Omron Sysmac Studio project 17-703_20171113_1 (Sysmac Studio 1.19.0.13, StandardProject)

# Controller new_Controller_0: NX1P2-9024DT version 1.13
Units and slaves: 節點1 : ASDA-A2-E CoE Drive (E001); 節點2 : ASDA-A2-E CoE Drive (E002)
Axis MC_Axis000, settings changed from default: AxisType=ServoType, FunctionLimit=SingleAxisPTP, UnitsConversion=EnumElement2, UnitsNumerator=1280000, UnitsDenominator=20, MaxVelocity=500, MaxJogVelocity=500, PositiveSoftwareLimit=305, HomingMode=BackupAndProximitySignalOn, StartDirection=NegativeDirection, HomingVelocity=50, HomingApproachVelocity=3, CompensationVelocity=1
Axis MC_Axis001, settings changed from default: AxisNumber=1, AxisType=ServoType, FunctionLimit=SingleAxisPTP, UnitsConversion=EnumElement2, UnitsNumerator=1280000, UnitsDenominator=20, MaxVelocity=500, MaxJogVelocity=500, PositiveSoftwareLimit=307, NegativeSoftwareLimit=-20, HomingMode=BackupAndProximitySignalOn, StartDirection=NegativeDirection, HomingVelocity=50, HomingApproachVelocity=3, CompensationVelocity=1
Task PrimaryTask (priority 4, period or condition 2000): prAxis, prConverter, prError, Postion_Control, PR_fix, 鎖付程式, 異常回0點, 系統初始, cycletime2, 原點復歸

TYPE stWorkPositionData : STRUCT
    ExPosition_X : array[0..10,0..10] of LREAL;  (* X軸鎖付位置 *)
    ExPosition_Y : array[0..10,0..10] of LREAL;  (* Y軸鎖付位置 *)
    ScrewData : array[0..10,0..10] of INT;  (* 鎖組別 *)
    Name_Data : array[0..10] of STRING[16];  (* 機種名稱 *)
    SV_AbsSpeed_X : array[0..10,0..10] of LREAL;  (* 伺服X_ABS速度32 *)
    SV_AbsSpeed_Y : array[0..10,0..10] of LREAL;  (* 伺服Y_ABS速度32 *)
    FinialPoint : array[0..10,0..10] of BOOL;
END_STRUCT END_TYPE
TYPE stAxis : STRUCT
    pbServoOn : BOOL;
    pbReset : BOOL;
    pbSerchHome : BOOL;  (* 原點搜尋開關 *)
    pbJOGForward : BOOL;  (* 手動前進 *)
    pbJOGBackward : BOOL;  (* 手動後退 *)
    pbStop : BOOL;
    pbMoveAbs : BOOL;  (* 自動移位開始 *)
    bMoveAbsDone : BOOL;  (* 到達位置 *)
    bHoming : BOOL;  (* 原點搜尋中 *)
    bServoOn : BOOL;
    bAtTHMoveSavePosition : BOOL;
    lrCurrentPosition : LREAL;  (* 現在位置 *)
    lrMoveAbsAddData : LREAL;  (* 自動移動位置 *)
    lrMoveAbsVelocity : LREAL;  (* 自動移動速度 *)
    lrMoveJogVelocity : LREAL;  (* 手動移動速度 *)
END_STRUCT END_TYPE

VAR_GLOBAL
    PB_Reset : BOOL;  (* 停止復歸開關; at BuiltInIO://cpu/#0/Input_Bit_01; published *)
    PB_Start : BOOL;  (* 啟動開關; at BuiltInIO://cpu/#0/Input_Bit_00; published *)
    PB_EStop : BOOL;  (* 急停開關; at BuiltInIO://cpu/#0/Input_Bit_02; published *)
    LS_UpDownBack : BOOL;  (* 鎖螺絲歸; at BuiltInIO://cpu/#0/Input_Bit_03; published *)
    LS_UpDownOut : BOOL;  (* 鎖螺絲出; at BuiltInIO://cpu/#0/Input_Bit_04; published *)
    LS_FixBack : BOOL;  (* 壓制歸; at BuiltInIO://cpu/#0/Input_Bit_05; published *)
    LS_FixOut : BOOL;  (* 壓制出; at BuiltInIO://cpu/#0/Input_Bit_06; published *)
    SNR_AirSource : BOOL;  (* 入氣源; at BuiltInIO://cpu/#0/Input_Bit_07; published *)
    SNR_CheckBody : BOOL;  (* 本體檢知; at BuiltInIO://cpu/#0/Input_Bit_08; published *)
    SNR_GratingUP : BOOL;  (* 安全光柵上; at BuiltInIO://cpu/#0/Input_Bit_09; published *)
    SNR_GratingDown : BOOL;  (* 安全光柵下; at BuiltInIO://cpu/#0/Input_Bit_10; published *)
    Check_GratingUP : BOOL;  (* 光柵自我檢測上; at BuiltInIO://cpu/#0/Input_Bit_11; published *)
    Check_GratingDown : BOOL;  (* 光柵自我檢測下; at BuiltInIO://cpu/#0/Input_Bit_12; published *)
    SNR_Float : BOOL;  (* 浮瑣檢知; at BuiltInIO://cpu/#0/Input_Bit_13; published *)
    SOL_FixBack : BOOL;  (* 壓制; at BuiltInIO://cpu/#0/Output_Bit_00; published *)
    SOL_UpDownBack : BOOL;  (* 鎖付上下; at BuiltInIO://cpu/#0/Output_Bit_01; published *)
    BZ : BOOL;  (* at BuiltInIO://cpu/#0/Output_Bit_02; published *)
    YL : BOOL;  (* at BuiltInIO://cpu/#0/Output_Bit_03; published *)
    GL : BOOL;  (* at BuiltInIO://cpu/#0/Output_Bit_04; published *)
    RL : BOOL;  (* at BuiltInIO://cpu/#0/Output_Bit_05; published *)
    NameTestData AT %w400 : ARRAY[0..1] OF STRING[16];
    SOL_FixOut : BOOL;  (* at BuiltInIO://cpu/#0/Output_Bit_06; published *)
    SOL_UpDownOut : BOOL;  (* at BuiltInIO://cpu/#0/Output_Bit_07; published *)
    Servo_OUT_Ready : BOOL;  (* 日東準備; at IOBus://unit#2/Input Bit 16 bits/Input Bit 00; published *)
    Servo_OUT_OK : BOOL;  (* 日東鎖付OK; at IOBus://unit#2/Input Bit 16 bits/Input Bit 01; published *)
    Servo_OUT_NOK : BOOL;  (* 日東鎖付NG; at IOBus://unit#2/Input Bit 16 bits/Input Bit 02; published *)
    Servo_OUT_Error : BOOL;  (* 日東異常; at IOBus://unit#2/Input Bit 16 bits/Input Bit 03; published *)
    Servo_OUT_Fioat : BOOL;  (* 日東鎖螺絲浮鎖測試OK; at IOBus://unit#2/Input Bit 16 bits/Input Bit 04; published *)
    Servo_OUT_Start : BOOL;  (* 日東同期鎖付啟動; at IOBus://unit#2/Input Bit 16 bits/Input Bit 05; published *)
    Servo_OUT_Angle : BOOL;  (* 日東角度判定OK; at IOBus://unit#2/Input Bit 16 bits/Input Bit 06; published *)
    Servo_OUT_Wave_AX1 : BOOL;  (* 日東波形處理OK; at IOBus://unit#2/Input Bit 16 bits/Input Bit 07; published *)
    Servo_IN_Start : BOOL;  (* 日東啟動; at IOBus://unit#3/Output Bit 8 bits/Output Bit 00; published *)
    Servo_IN_TorqueBit0 : BOOL;  (* 日東工作選擇0; at IOBus://unit#3/Output Bit 8 bits/Output Bit 01; published *)
    Servo_IN_TorqueBit1 : BOOL;  (* 日東工作選擇1; at IOBus://unit#3/Output Bit 8 bits/Output Bit 02; published *)
    Servo_IN_TorqueBit2 : BOOL;  (* 日東工作選擇2; at IOBus://unit#3/Output Bit 8 bits/Output Bit 03; published *)
    Servo_IN_TorqueBit3 : BOOL;  (* 日東工作選擇3; at IOBus://unit#3/Output Bit 8 bits/Output Bit 04; published *)
    Servo_IN_output : BOOL;  (* 日東外部信號; at IOBus://unit#3/Output Bit 8 bits/Output Bit 05; published *)
    Servo_IN_ALLStart : BOOL;  (* 日東同期鎖付啟動; at IOBus://unit#3/Output Bit 8 bits/Output Bit 06; published *)
END_VAR
VAR_GLOBAL CONSTANT
    MC_Axis000 : _sAXIS_REF;  (* at MC://_MC_AX[0] *)
    MC_Axis001 : _sAXIS_REF;  (* at MC://_MC_AX[1] *)
END_VAR
VAR_GLOBAL
    Ax_X : stAxis;
    Ax_Y : stAxis;
END_VAR
VAR_GLOBAL RETAIN
    WorkPositionData : stWorkPositionData;  (* published *)
END_VAR
VAR_GLOBAL
    SystemReadyStatus : BOOL;  (* published *)
    MachineRun : BOOL;  (* published *)
    ErrorStatus_MachineStop : BOOL;  (* 機器停機異常; published *)
    ErrorStatus_MachineNonStop : BOOL;  (* 機器不停機異常; published *)
    Manual2AutoFlag : BOOL;  (* published *)
    AutoStatus AT %W000.00 : BOOL;  (* 自動狀態; published *)
    PB_UpDownBack AT %W000.01 : BOOL;  (* 手動鎖付上; published *)
    PB_UpDownOut AT %W000.02 : BOOL;  (* 手動鎖付下; published *)
    PB_FixBack AT %W000.03 : BOOL;  (* 手動壓制回; published *)
    PB_FixOut AT %W000.04 : BOOL;  (* 手動壓制出; published *)
    PB_ScrewStart AT %W000.05 : BOOL;  (* published *)
    PB_ServoY_Back AT %W000.06 : BOOL;  (* 手動伺服Y回; published *)
    PB_ServoY_Out AT %W000.07 : BOOL;  (* 手動伺服Y出; published *)
    PB_ServoX_Back AT %W000.08 : BOOL;  (* 手動伺服X回; published *)
    PB_ServoX_Out AT %W000.09 : BOOL;  (* 手動伺服X出; published *)
    PB_ServoOn_X AT %W000.10 : BOOL;  (* 手動伺服X_ServoON; published *)
    PB_ServoOn_Y AT %W000.11 : BOOL;  (* 手動伺服Y_ServoON; published *)
    PB_SetPostion AT %W000.12 : BOOL;  (* 位置設定開關; published *)
    PB_FinalPoint AT %W000.13 : BOOL;  (* 最終點設定開關; published *)
    PB_PostionGo AT %W000.14 : BOOL;  (* 點位啟動; published *)
    PB_Set_Homed AT %W000.15 : BOOL;  (* 伺服回原點開關; published *)
    PB_HMI_RESRT AT %W001.00 : BOOL;  (* published *)
    State_Homed_MC AT %W001.01 : BOOL;  (* 伺服原點; published *)
    State_Homing_MC AT %W001.02 : BOOL;  (* 伺服回原點中; published *)
    State_HomeSerching_X AT %W001.03 : BOOL;  (* X伺服回原點中; published *)
    State_Homed_X AT %W001.04 : BOOL;  (* X伺服原點; published *)
    State_HomeSerching_Y AT %W001.05 : BOOL;  (* Y伺服回原點中; published *)
    State_Homed_Y AT %W001.06 : BOOL;  (* Y伺服原點; published *)
    ScrewStartStatus AT %W001.07 : BOOL;  (* published *)
    LS_FixOut1 AT %W001.15 : BOOL;  (* published *)
    HMI_ScrewOK1 AT %W002.00 : BOOL;  (* published *)
    HMI_ScrewOK2 AT %W002.01 : BOOL;  (* published *)
    LS_FixBack1 AT %W001.14 : BOOL;  (* published *)
    LS_UpDownBack1 AT %W001.12 : BOOL;  (* published *)
    PB_HMI_SetScrew AT %w001.11 : BOOL;  (* published *)
    LS_UpDownOut1 AT %W001.13 : BOOL;  (* published *)
    PB_HMI_BzStpo AT %w001.10 : BOOL;  (* published *)
    ScrewFinish AT %W001.08 : BOOL;  (* published *)
    HMI_Servo_IN_Start AT %W001.09 : BOOL;  (* published *)
END_VAR
VAR_GLOBAL RETAIN
    SV_ServoXJogSpeed : LREAL;  (* 設定伺服X_JOG速度64; published *)
    SV_ServoYJogSpeed : LREAL;  (* 設定伺服Y_JOG速度64; published *)
    SV_ServoXJogSpeed_R AT %D000 : REAL;  (* 設定伺服X_JOG速度32; published *)
    SV_ServoYJogSpeed_R AT %D002 : REAL;  (* 設定伺服Y_JOG速度32; published *)
    SV_AbsSpeedX_R AT %D004 : REAL;  (* 設定伺服X_ABS速度32; published *)
    SV_AbsSpeedY_R AT %D006 : REAL;  (* 設定伺服Y_ABS速度32; published *)
    HMI_SV_AbsSpeedX_R AT %D008 : REAL;  (* 顯示伺服X_ABS速度32; published *)
    HMI_SV_AbsSpeedY_R AT %D010 : REAL;  (* 顯示伺服Y_ABS速度32; published *)
    HMI_SV_CurrentPositionX AT %D012 : REAL;  (* 人機現在位置X顯示; published *)
    HMI_SV_CurrentPositionY AT %D014 : REAL;  (* 人機現在位置Y顯示; published *)
    Type_Data AT %D042 : INT;  (* 設定組別; published *)
    PointData AT %D043 : INT;  (* 設定點位; published *)
    Screw_Data1 AT %D044 : INT;  (* 設定鎖付值; published *)
    Screw_Data2 AT %D045 : INT;
    Screw_Data3 AT %D046 : INT;
    Screw_Data4 AT %D047 : INT;
    OK_Count AT %D050 : DINT;  (* published *)
    AllOK_Count AT %D052 : DINT;  (* published *)
    HMISV_CycleTime1 AT %D054 : DINT;  (* published *)
    HMISV_CycleTime2 AT %D056 : DINT;  (* published *)
END_VAR
VAR_GLOBAL
    HMI_Name : ARRAY[0..10] OF STRING[32];  (* 顯示已設定組別名稱; published *)
    HMI_ScrewOK3 AT %W002.02 : BOOL;  (* published *)
    HMI_ScrewOK4 AT %W002.03 : BOOL;  (* published *)
END_VAR
VAR_GLOBAL RETAIN
    HMI_Name1 AT %D200 : STRING[16];  (* published *)
    HMI_Name2 AT %D208 : STRING[16];  (* published *)
    HMI_Name3 AT %D216 : STRING[16];  (* published *)
    HMI_Name4 AT %D224 : STRING[16];  (* published *)
    HMI_Name5 AT %D232 : STRING[16];  (* published *)
    HMI_Name6 AT %D240 : STRING[16];  (* published *)
    HMI_Name7 AT %D248 : STRING[16];  (* published *)
    HMI_Name8 AT %D256 : STRING[16];  (* published *)
    HMI_Name9 AT %D264 : STRING[16];  (* published *)
    HMI_Name10 AT %D272 : STRING[16];  (* published *)
END_VAR
VAR_GLOBAL
    HMI_SV_Name AT %W360 : STRING[16];  (* published *)
    HMI_ScrewNG1 AT %W002.04 : BOOL;  (* published *)
    HMI_ScrewNG2 AT %W002.05 : BOOL;  (* published *)
    HMI_ScrewNG3 AT %W002.06 : BOOL;  (* published *)
    HMI_ScrewNG4 AT %W002.07 : BOOL;  (* published *)
    HMI_Float1 AT %W002.08 : BOOL;  (* published *)
    HMI_SV_Screw_Data4 AT %W153 : INT;
    HMI_SV_Screw_Data3 AT %W152 : INT;
    HMI_SV_Screw_Data2 AT %W151 : INT;
    HMI_SV_Screw_Data1 AT %W150 : INT;
    HMI_SV_Screw_Data AT %W104 : INT;  (* 顯示現在鎖付值; published *)
    HMI_PositionY AT %W102 : REAL;  (* 顯示已設定位置Y顯示; published *)
    HMI_PositionX AT %W100 : REAL;  (* 顯示已設定位置X顯示; published *)
    HMI_Float2 AT %W002.09 : BOOL;  (* published *)
    HMI_Float4 AT %W002.11 : BOOL;  (* published *)
    HMI_SVFinalPoint AT %W002.12 : BOOL;  (* HMI最終點顯示; published *)
    PB_ResetOk_Count AT %W002.13 : BOOL;  (* published *)
    PB_Name_Set AT %w002.14 : BOOL;  (* published *)
    HMI_Float3 AT %W002.10 : BOOL;  (* published *)
END_VAR
VAR_GLOBAL RETAIN
    Screw_OK : ARRAY[0..10] OF BOOL;  (* published *)
    Screw_NG : ARRAY[0..10] OF BOOL;  (* published *)
    Screw_Float : ARRAY[0..10] OF BOOL;  (* published *)
END_VAR
VAR_GLOBAL
    Error_LS_UpDownBack AT %W200.00 : BOOL;  (* published *)
    Error_LS_UpDownOut AT %W200.01 : BOOL;  (* published *)
    Error_LS_FixBack AT %W200.02 : BOOL;  (* published *)
    Error_LS_FixOut AT %W200.03 : BOOL;  (* published *)
    Error_Check_GratingUP AT %W200.04 : BOOL;  (* 光柵自我檢測上異常; published *)
    Error_Check_GratingDown AT %W200.05 : BOOL;  (* 光柵自我檢測下異常; published *)
    Error_GratingUP AT %W200.06 : BOOL;  (* 光柵上異常; published *)
    Error_GratingDown AT %W200.07 : BOOL;  (* 光柵下異常; published *)
    Error_EStopPB AT %W200.08 : BOOL;  (* published *)
    Error_ChangeBodyNG AT %W200.14 : BOOL;  (* published *)
    Error_ScrewNG AT %W200.13 : BOOL;  (* published *)
    Error_SNR_CheckBody AT %W200.12 : BOOL;  (* published *)
    Error_SNR_AirSource AT %W200.11 : BOOL;  (* published *)
    Error_Servo_Y AT %W200.10 : BOOL;  (* 伺服異常Y; published *)
    Error_Servo_X AT %W200.09 : BOOL;  (* 伺服異常X; published *)
    Error_LS_Status : BOOL;  (* 磁簧開關異常; published *)
    Error_Grating_Status : BOOL;  (* published *)
    Error_Status : BOOL;  (* published *)
    Error_Servo : BOOL;  (* published *)
    XN_OT : BOOL;  (* published *)
    XP_OT : BOOL;  (* published *)
    YN_OT : BOOL;  (* published *)
    YP_OT : BOOL;  (* published *)
    MachineRunStatus : BOOL;
    HMI_LT_ServoRuning AT %W003.01 : BOOL;  (* published *)
    HMI_LT_ServoFinish AT %w003.00 : BOOL;  (* published *)
    LT_ServoFinish1 AT %w003.02 : BOOL;  (* published *)
    LT_ServoFinish2 AT %w003.04 : BOOL;  (* published *)
    LT_ServoRuning1 AT %w003.05 : BOOL;  (* published *)
    LT_ServoRuning2 AT %w003.06 : BOOL;  (* published *)
    Error_XP_OT AT %W200.15 : BOOL;  (* published *)
    Error_XN_OT AT %W201.00 : BOOL;  (* published *)
    Error_YP_OT AT %W201.01 : BOOL;  (* published *)
    Error_YN_OT AT %W201.02 : BOOL;  (* published *)
END_VAR
VAR_GLOBAL RETAIN
    Screw_Data5 AT %D060 : INT;  (* published *)
    Screw_Data6 AT %D061 : INT;  (* published *)
    Screw_Data7 AT %D062 : INT;  (* published *)
    Screw_Data8 AT %D063 : INT;  (* published *)
    Screw_Data9 AT %D064 : INT;  (* published *)
    Screw_Data10 AT %D065 : INT;  (* published *)
END_VAR
VAR_GLOBAL
    HMI_SV_Screw_Data5 AT %W154 : INT;  (* published *)
    HMI_SV_Screw_Data6 AT %W155 : INT;  (* published *)
    HMI_SV_Screw_Data7 AT %W156 : INT;  (* published *)
    HMI_SV_Screw_Data8 AT %W157 : INT;  (* published *)
    HMI_SV_Screw_Data9 AT %W158 : INT;  (* published *)
    HMI_SV_Screw_Data10 AT %W159 : INT;  (* published *)
    LS_ExternalStart : BOOL;  (* 外部可啟動信號; at IOBus://unit#2/Input Bit 16 bits/Input Bit 08; published *)
    HMI_SV_ReclaimerOK AT %w003.07 : BOOL;  (* 外部取料完成; published *)
END_VAR
VAR_GLOBAL RETAIN
    ReclaimerOK : BOOL;  (* published *)
END_VAR
VAR_GLOBAL
    Error_ReclaimerOK AT %W201.03 : BOOL;  (* 取料未完成異常; published *)
END_VAR
VAR_GLOBAL RETAIN
    PB_ExternalStart AT %H00.0 : BOOL;  (* published *)
END_VAR

PROGRAM prAxis
VAR
    MC_Power_Ax1 : MC_Power;
    MC_Power_Ax2 : MC_Power;
    MC_Home_Ax1 : MC_Home;
    MC_Home_Ax2 : MC_Home;
    MC_MoveJog_Ax1 : MC_MoveJog;
    MC_MoveJog_Ax2 : MC_MoveJog;
    MC_Reset_Ax1 : MC_Reset;
    MC_Reset_Ax2 : MC_Reset;
    MC_MoveAbsolute_Ax1 : MC_MoveAbsolute;
    MC_MoveAbsolute_Ax2 : MC_MoveAbsolute;
    MC_Stop_Ax1 : MC_Stop;
    MC_Stop_Ax2 : MC_Stop;
    XN_HOME : BOOL;
    Y_HOME : BOOL;
END_VAR
VAR_EXTERNAL CONSTANT
    MC_Axis001 : _sAXIS_REF;
END_VAR
VAR_EXTERNAL
    Ax_X : stAxis;
END_VAR
VAR_EXTERNAL CONSTANT
    MC_Axis000 : _sAXIS_REF;
END_VAR
VAR_EXTERNAL
    Ax_Y : stAxis;
    WorkPositionData : stWorkPositionData;
    PB_EStop : BOOL;
    Error_EStopPB : BOOL;
    PB_ServoOn_X : BOOL;
    PB_ServoOn_Y : BOOL;
    PB_Reset : BOOL;
    XP_OT : BOOL;
    XN_OT : BOOL;
    YN_OT : BOOL;
    YP_OT : BOOL;
    ErrorStatus_MachineStop : BOOL;
    LS_UpDownBack : BOOL;
    SOL_UpDownOut : BOOL;
    LS_UpDownBack1 : BOOL;
    SNR_AirSource : BOOL;
    SNR_GratingDown : BOOL;
    SNR_GratingUP : BOOL;
    Error_GratingUP : BOOL;
    Error_GratingDown : BOOL;
    Error_Grating_Status : BOOL;
    Error_XP_OT : BOOL;
    Error_YP_OT : BOOL;
    Error_YN_OT : BOOL;
END_VAR
(*X軸*)
//Servo on
Ax_X.pbServoOn:=PB_ServoOn_X;
MC_Power_Ax1(Axis:=MC_Axis000, Enable:=Ax_X.pbServoOn AND NOT(Error_EStopPB));
//Reset
MC_Reset_Ax1(Axis:=MC_Axis000, Execute:=Ax_X.pbReset);
//Home
MC_Home_Ax1(Axis:=MC_Axis000, Execute:=Ax_X.pbSerchHome AND Ax_X.bServoOn);
//STOP
MC_Stop_Ax1(Axis:=MC_Axis000, Execute:=Ax_X.pbStop);
//JOG
MC_MoveJog_Ax1(Axis:=MC_Axis000, PositiveEnable:=Ax_X.pbJOGForward , NegativeEnable:=Ax_X.pbJOGBackward , Velocity:=Ax_X.lrMoveJogVelocity,acceleration:=5000,deceleration:=5000);
//絕對定位
MC_MoveAbsolute_Ax1(Axis:=MC_Axis000, Execute:=Ax_X.pbMoveAbs AND Ax_X.bServoOn AND MC_Axis000.Details.Homed,
					Position:=Ax_X.lrMoveAbsAddData,	Velocity:=Ax_X.lrMoveAbsVelocity,acceleration:=5000,deceleration:=5000,
					Done=>Ax_X.bMoveAbsDone);

//定義
//Servo On
Ax_X.bServoOn:=MC_Axis000.DrvStatus.ServoOn;
//找HOME
Ax_X.bHoming:=MC_Axis000.Status.Homing;
//現在位置
Ax_X.lrCurrentPosition:=MC_Axis000.Act.Pos;
(*Y軸*)
//Servo on
Ax_Y.pbServoOn:=PB_ServoOn_Y;
MC_Power_Ax2(Axis:=MC_Axis001, Enable:=Ax_Y.pbServoOn AND NOT(Error_EStopPB));
//Reset
MC_Reset_Ax2(Axis:=MC_Axis001, Execute:=Ax_Y.pbReset);
//Home
MC_Home_Ax2(Axis:=MC_Axis001, Execute:=Ax_Y.pbSerchHome AND Ax_Y.bServoOn);
//STOP
MC_Stop_Ax2(Axis:=MC_Axis001, Execute:=Ax_Y.pbStop );
//JOG
MC_MoveJog_Ax2(Axis:=MC_Axis001, PositiveEnable:=Ax_Y.pbJOGForward  , NegativeEnable:=Ax_Y.pbJOGBackward  , Velocity:=Ax_Y.lrMoveJogVelocity,acceleration:=5000,deceleration:=5000);
//絕對定位
MC_MoveAbsolute_Ax2(Axis:=MC_Axis001, Execute:=Ax_Y.pbMoveAbs AND Ax_Y.bServoOn AND MC_Axis001.Details.Homed,
					Position:=Ax_Y.lrMoveAbsAddData,	Velocity:=Ax_Y.lrMoveAbsVelocity,acceleration:=5000,deceleration:=5000,
					Done=>Ax_Y.bMoveAbsDone);

//定義
//Servo On
Ax_Y.bServoOn:=MC_Axis001.DrvStatus.ServoOn;
//找HOME
Ax_Y.bHoming:=MC_Axis001.Status.Homing;
//現在位置
Ax_Y.lrCurrentPosition:=MC_Axis001.Act.Pos;

//RESET
Ax_X.pbReset:=PB_Reset;
Ax_Y.pbReset:=PB_Reset;
//Stop
Ax_X.pbStop:= NOT(PB_EStop) OR Error_Grating_Status;
Ax_Y.pbStop:= NOT(PB_EStop) OR Error_Grating_Status;
XN_OT:=MC_Axis000.DrvStatus.N_OT;
XP_OT:=MC_Axis000.DrvStatus.P_OT;
YN_OT:=MC_Axis001.DrvStatus.N_OT;
YP_OT:=MC_Axis001.DrvStatus.P_OT;
XN_HOME:=MC_Axis000.DrvStatus.HomeSw;
Y_HOME:=MC_Axis001.DrvStatus.HomeSw;
END_PROGRAM

PROGRAM prConverter
VAR
    Status_FinalPoint : BOOL;
    R_TRIG_1 : R_TRIG;
END_VAR
VAR_EXTERNAL
    SV_ServoXJogSpeed : LREAL;
    SV_AbsSpeedX_R : REAL;
    SV_ServoXJogSpeed_R : REAL;
    SV_ServoYJogSpeed : LREAL;
    SV_ServoYJogSpeed_R : REAL;
    Ax_X : stAxis;
    Type_Data : INT;
    PointData : INT;
    WorkPositionData : stWorkPositionData;
    SV_AbsSpeedY_R : REAL;
    State_Homed_X : BOOL;
END_VAR
VAR_EXTERNAL CONSTANT
    MC_Axis000 : _sAXIS_REF;
END_VAR
VAR_EXTERNAL
    State_Homed_Y : BOOL;
END_VAR
VAR_EXTERNAL CONSTANT
    MC_Axis001 : _sAXIS_REF;
END_VAR
VAR_EXTERNAL
    State_HomeSerching_X : BOOL;
    State_HomeSerching_Y : BOOL;
    Ax_Y : stAxis;
    State_Homed_MC : BOOL;
    State_Homing_MC : BOOL;
    PB_SetPostion : BOOL;
    PB_FinalPoint : BOOL;
    HMI_SV_CurrentPositionX : REAL;
    HMI_SV_CurrentPositionY : REAL;
    HMI_PositionX : REAL;
    HMI_PositionY : REAL;
    HMI_SVFinalPoint : BOOL;
    AutoStatus : BOOL;
    HMI_SV_Screw_Data : INT;
    HMI_SV_AbsSpeedX_R : REAL;
    HMI_SV_AbsSpeedY_R : REAL;
    HMI_ScrewNG1 : BOOL;
    Screw_NG : ARRAY[0..10] OF BOOL;
    HMI_ScrewNG2 : BOOL;
    HMI_ScrewNG3 : BOOL;
    HMI_ScrewNG4 : BOOL;
    HMI_ScrewOK1 : BOOL;
    Screw_OK : ARRAY[0..10] OF BOOL;
    HMI_ScrewOK2 : BOOL;
    HMI_ScrewOK3 : BOOL;
    HMI_ScrewOK4 : BOOL;
    HMI_Name1 : STRING[16];
    HMI_Name2 : STRING[16];
    HMI_Name3 : STRING[16];
    HMI_Name4 : STRING[16];
    HMI_Name5 : STRING[16];
    HMI_Name6 : STRING[16];
    HMI_Name7 : STRING[16];
    HMI_Name8 : STRING[16];
    HMI_Name9 : STRING[16];
    HMI_Name10 : STRING[16];
    HMI_Name : ARRAY[0..10] OF STRING[32];
    PB_Name_Set : BOOL;
    Screw_Data1 : INT;
    Screw_Data2 : INT;
    Screw_Data3 : INT;
    Screw_Data4 : INT;
    HMI_SV_Screw_Data1 : INT;
    HMI_SV_Screw_Data4 : INT;
    HMI_SV_Screw_Data3 : INT;
    HMI_SV_Screw_Data2 : INT;
    PB_HMI_SetScrew : BOOL;
    HMI_SV_Name : STRING[16];
    HMISV_CycleTime1 : DINT;
    NameTestData : ARRAY[0..1] OF STRING[16];
    Screw_Data10 : INT;
    Screw_Data9 : INT;
    Screw_Data5 : INT;
    Screw_Data6 : INT;
    Screw_Data7 : INT;
    Screw_Data8 : INT;
    HMI_SV_Screw_Data10 : INT;
    HMI_SV_Screw_Data9 : INT;
    HMI_SV_Screw_Data8 : INT;
    HMI_SV_Screw_Data7 : INT;
    HMI_SV_Screw_Data6 : INT;
    HMI_SV_Screw_Data5 : INT;
    HMI_SV_ReclaimerOK : BOOL;
    ReclaimerOK : BOOL;
    LS_ExternalStart : BOOL;
    Screw_Float : ARRAY[0..10] OF BOOL;
    HMI_Float2 : BOOL;
    HMI_Float3 : BOOL;
    HMI_Float4 : BOOL;
    HMI_Float1 : BOOL;
END_VAR
SV_ServoXJogSpeed:=REAL_TO_LREAL(SV_ServoXJogSpeed_R);//X軸手動速度單位轉換
SV_ServoYJogSpeed:=REAL_TO_LREAL(SV_ServoYJogSpeed_R);//Y軸手動速度單位轉換
State_Homed_X:=MC_Axis000.Details.Homed;//X軸復歸完成
State_Homed_Y:=MC_Axis001.Details.Homed;//Y軸復歸完成
State_HomeSerching_X:=Ax_X.bHoming;//X軸復歸中
State_HomeSerching_Y:=Ax_Y.bHoming;//Y軸復歸中
State_Homed_MC:=State_Homed_X AND State_Homed_Y AND NOT(State_Homing_MC);//原點復歸完成
State_Homing_MC:=State_HomeSerching_X OR State_HomeSerching_Y;//原點復歸中
//位置_鎖付組別寫入
IF PB_SetPostion THEN
	WorkPositionData.ExPosition_X[Type_Data,PointData]:=Ax_X.lrCurrentPosition;
    WorkPositionData.ExPosition_Y[Type_Data,PointData]:=Ax_Y.lrCurrentPosition;
	WorkPositionData.SV_AbsSpeed_X[Type_Data,PointData]:=REAL_TO_LREAL(SV_AbsSpeedX_R);
    WorkPositionData.SV_AbsSpeed_Y[Type_Data,PointData]:=REAL_TO_LREAL(SV_AbsSpeedY_R);
END_IF;

//最終點寫入
R_TRIG_1(Clk:=PB_FinalPoint);
IF R_TRIG_1.Q AND NOT(Status_FinalPoint)  THEN
	WorkPositionData.FinialPoint[Type_Data,PointData]:=TRUE;
END_IF;
//最終點取消
IF R_TRIG_1.Q AND Status_FinalPoint  THEN
	WorkPositionData.FinialPoint[Type_Data,PointData]:=FALSE;
END_IF;
Status_FinalPoint:=WorkPositionData.FinialPoint[Type_Data,PointData];

//現在位置HMI
HMI_SV_CurrentPositionX:=LREAL_TO_REAL(Ax_X.lrCurrentPosition);
HMI_SV_CurrentPositionY:=LREAL_TO_REAL(Ax_Y.lrCurrentPosition);
//設定位置
HMI_PositionX:=LREAL_TO_REAL(WorkPositionData.ExPosition_X[Type_Data,PointData]);
HMI_PositionY:=LREAL_TO_REAL(WorkPositionData.ExPosition_Y[Type_Data,PointData]);
//最終點顯示
HMI_SVFinalPoint:=WorkPositionData.FinialPoint[Type_Data,PointData];
//人機顯示
HMI_SV_AbsSpeedX_R:=LREAL_TO_REAL(WorkPositionData.SV_AbsSpeed_X[Type_Data,PointData]);
HMI_SV_AbsSpeedY_R:=LREAL_TO_REAL(WorkPositionData.SV_AbsSpeed_Y[Type_Data,PointData]);
//HMI_Name[Type_Data]:=WorkPositionData.Name_Data[Type_Data];
HMI_SV_Name:=WorkPositionData.Name_Data[Type_Data];
NameTestData[0]:=HMI_SV_Name;
HMI_ScrewNG1:=Screw_NG[1];
HMI_ScrewNG2:=Screw_NG[2];
HMI_ScrewNG3:=Screw_NG[3];
HMI_ScrewNG4:=Screw_NG[4];
HMI_ScrewOK1:=Screw_OK[1];
HMI_ScrewOK2:=Screw_OK[2];
HMI_ScrewOK3:=Screw_OK[3];
HMI_ScrewOK4:=Screw_OK[4];
HMI_Float1:=Screw_Float[1];
HMI_Float2:=Screw_Float[2];
HMI_Float3:=Screw_Float[3];
HMI_Float4:=Screw_Float[4];
IF PB_Name_Set THEN
WorkPositionData.Name_Data[1]:=HMI_Name1;
WorkPositionData.Name_Data[2]:=HMI_Name2;
WorkPositionData.Name_Data[3]:=HMI_Name3;
WorkPositionData.Name_Data[4]:=HMI_Name4;
WorkPositionData.Name_Data[5]:=HMI_Name5;
WorkPositionData.Name_Data[6]:=HMI_Name6;
WorkPositionData.Name_Data[7]:=HMI_Name7;
WorkPositionData.Name_Data[8]:=HMI_Name8;
WorkPositionData.Name_Data[9]:=HMI_Name9;
WorkPositionData.Name_Data[10]:=HMI_Name10;
END_IF;
//日東組別寫入
IF PB_HMI_SetScrew THEN
WorkPositionData.ScrewData[Type_Data,1]:=Screw_Data1;
WorkPositionData.ScrewData[Type_Data,2]:=Screw_Data2;
WorkPositionData.ScrewData[Type_Data,3]:=Screw_Data3;
WorkPositionData.ScrewData[Type_Data,4]:=Screw_Data4;
WorkPositionData.ScrewData[Type_Data,5]:=Screw_Data5;
WorkPositionData.ScrewData[Type_Data,6]:=Screw_Data6;
WorkPositionData.ScrewData[Type_Data,7]:=Screw_Data7;
WorkPositionData.ScrewData[Type_Data,8]:=Screw_Data8;
WorkPositionData.ScrewData[Type_Data,9]:=Screw_Data9;
WorkPositionData.ScrewData[Type_Data,10]:=Screw_Data10;
END_IF;

//日東組別顯示
HMI_SV_Screw_Data:=WorkPositionData.ScrewData[Type_Data,PointData];
HMI_SV_Screw_Data1:=WorkPositionData.ScrewData[Type_Data,1];
HMI_SV_Screw_Data2:=WorkPositionData.ScrewData[Type_Data,2];
HMI_SV_Screw_Data3:=WorkPositionData.ScrewData[Type_Data,3];
HMI_SV_Screw_Data4:=WorkPositionData.ScrewData[Type_Data,4];
HMI_SV_Screw_Data5:=WorkPositionData.ScrewData[Type_Data,5];
HMI_SV_Screw_Data6:=WorkPositionData.ScrewData[Type_Data,6];
HMI_SV_Screw_Data7:=WorkPositionData.ScrewData[Type_Data,7];
HMI_SV_Screw_Data8:=WorkPositionData.ScrewData[Type_Data,8];
HMI_SV_Screw_Data9:=WorkPositionData.ScrewData[Type_Data,9];
HMI_SV_Screw_Data10:=WorkPositionData.ScrewData[Type_Data,10];
//外部取料信號顯示
HMI_SV_ReclaimerOK:=ReclaimerOK;	
END_PROGRAM

PROGRAM prError
VAR
    TON1 : ARRAY[0..10] OF TON;
    ExternalStart_status : BOOL;
    R_TRIG_1 : R_TRIG;
    R_TRIG_2 : R_TRIG;
    F_TRIG_1 : R_TRIG;
    F_TRIG_2 : F_TRIG;
END_VAR
VAR_EXTERNAL
    AutoStatus : BOOL;
    PB_Reset : BOOL;
    LS_UpDownBack : BOOL;
    SOL_UpDownBack : BOOL;
    LS_UpDownOut : BOOL;
    Error_LS_UpDownBack : BOOL;
    SOL_UpDownOut : BOOL;
    Error_LS_UpDownOut : BOOL;
    SOL_FixBack : BOOL;
    LS_FixBack : BOOL;
    Error_LS_FixBack : BOOL;
    LS_FixOut : BOOL;
    SOL_FixOut : BOOL;
    Error_LS_FixOut : BOOL;
    Error_EStopPB : BOOL;
    PB_EStop : BOOL;
END_VAR
VAR_EXTERNAL CONSTANT
    MC_Axis000 : _sAXIS_REF;
END_VAR
VAR_EXTERNAL
    Error_Servo_X : BOOL;
END_VAR
VAR_EXTERNAL CONSTANT
    MC_Axis001 : _sAXIS_REF;
END_VAR
VAR_EXTERNAL
    Error_Servo_Y : BOOL;
    Check_GratingUP : BOOL;
    Error_Check_GratingUP : BOOL;
    Check_GratingDown : BOOL;
    Error_Check_GratingDown : BOOL;
    SystemReadyStatus : BOOL;
    MachineRun : BOOL;
    SNR_GratingUP : BOOL;
    Error_GratingUP : BOOL;
    SNR_GratingDown : BOOL;
    Error_GratingDown : BOOL;
    SNR_AirSource : BOOL;
    Error_SNR_AirSource : BOOL;
    ErrorStatus_MachineStop : BOOL;
    Error_LS_Status : BOOL;
    Error_Servo : BOOL;
    Servo_OUT_Error : BOOL;
    Error_Grating_Status : BOOL;
    SNR_CheckBody : BOOL;
    Error_SNR_CheckBody : BOOL;
    PB_HMI_RESRT : BOOL;
    MachineRunStatus : BOOL;
    Screw_NG : ARRAY[0..10] OF BOOL;
    Error_ScrewNG : BOOL;
    LS_UpDownBack1 : BOOL;
    LS_UpDownOut1 : BOOL;
    LS_FixBack1 : BOOL;
    LS_FixOut1 : BOOL;
    Servo_IN_ALLStart : BOOL;
    Servo_IN_Start : BOOL;
    HMI_Servo_IN_Start : BOOL;
    ScrewFinish : BOOL;
    Error_ChangeBodyNG : BOOL;
    PB_Start : BOOL;
    Ax_X : stAxis;
    Ax_Y : stAxis;
    HMI_LT_ServoFinish : BOOL;
    LT_ServoFinish1 : BOOL;
    LT_ServoFinish2 : BOOL;
    HMI_LT_ServoRuning : BOOL;
    LT_ServoRuning1 : BOOL;
    LT_ServoRuning2 : BOOL;
    Type_Data : INT;
    WorkPositionData : stWorkPositionData;
    XP_OT : BOOL;
    Error_XP_OT : BOOL;
    PB_ServoOn_X : BOOL;
    XN_OT : BOOL;
    YP_OT : BOOL;
    Error_YP_OT : BOOL;
    PB_ServoOn_Y : BOOL;
    YN_OT : BOOL;
    Error_YN_OT : BOOL;
    Error_XN_OT : BOOL;
    State_Homed_MC : BOOL;
    LS_ExternalStart : BOOL;
    ReclaimerOK : BOOL;
    Error_ReclaimerOK : BOOL;
    PB_ExternalStart : BOOL;
    Screw_Float : ARRAY[0..10] OF BOOL;
END_VAR
IF AutoStatus AND NOT(PB_Reset) AND Type_Data<10  THEN
    TON1[0](In:=((SOL_UpDownBack AND NOT(LS_UpDownBack)) OR (NOT(LS_UpDownBack)  AND NOT(LS_UpDownOut) ) ), PT:=T#2s);
 (*上下歸異常磁簧開關*)
   IF TON1[0].Q THEN
	   Error_LS_UpDownBack:=TRUE;
   END_IF;
   IF LS_UpDownBack THEN
	   SOL_UpDownBack:=FALSE;
   END_IF;
  TON1[1](In:=((SOL_UpDownOut AND NOT(LS_UpDownOut)) OR (NOT(LS_UpDownBack) AND NOT(LS_UpDownOut) )  ), PT:=T#2s);
  (*上下出異常磁簧開關*)
   IF TON1[1].Q THEN
	   Error_LS_UpDownOut:=TRUE;
   END_IF;
   IF LS_UpDownOut THEN
	   SOL_UpDownOut:=FALSE;
   END_IF;
   TON1[2](In:=((SOL_FixBack AND NOT(LS_FixBack)) OR (NOT(LS_FixBack) AND NOT(LS_FixOut) )  ), PT:=T#2s);
 (*壓制歸異常磁簧開關*)
   IF TON1[2].Q THEN
	   Error_LS_FixBack:=TRUE;
   END_IF;
   IF LS_FixBack THEN
	   SOL_FixBack:=FALSE;
   END_IF;
TON1[3](In:=((SOL_FixOut AND NOT(LS_FixOut)) OR (NOT(LS_FixBack) AND NOT(LS_FixOut) ) ), PT:=T#2s);
(*壓制出異常磁簧開關*)
   IF TON1[3].Q THEN
	   Error_LS_FixOut:=TRUE;
   END_IF;
   IF LS_FixOut THEN
	   SOL_FixOut:=FALSE;
   END_IF;
END_IF;

//ESTOP
TON1[4](In:=P_On , PT:=T#100ms);
IF TON1[4].Q AND NOT(PB_EStop)   THEN
	Error_EStopPB:=TRUE;
END_IF;

//氣壓源異常
IF NOT(SNR_AirSource) AND TON1[4].Q THEN
	Error_SNR_AirSource:=TRUE;
END_IF;

//SERVO
IF MC_Axis000.DrvStatus.DrvAlarm AND TON1[4].Q THEN
	Error_Servo_X:=TRUE;
END_IF;
IF MC_Axis001.DrvStatus.DrvAlarm AND TON1[4].Q THEN
	Error_Servo_Y:=TRUE;
END_IF;

//本體異常
R_TRIG_1(Clk:=MachineRun);
IF R_TRIG_1.Q AND NOT(SNR_CheckBody) AND NOT(Type_Data=10) THEN
	Error_SNR_CheckBody:=TRUE;
END_IF;

//光閘自我檢測異常(上)
//IF NOT(Check_GratingUP) AND TON1[4].Q  THEN
//	Error_Check_GratingUP:=TRUE;
//END_IF;

//光閘自我檢測異常(下)
//IF NOT(Check_GratingDown) AND TON1[4].q  THEN
//	Error_Check_GratingDown:=TRUE;
//END_IF;

//運轉中光閘異常(上)
IF MachineRun AND NOT(SNR_GratingUP) THEN
	Error_GratingUP:=TRUE;
END_IF;

//運轉中光閘異常(下)
IF MachineRun AND NOT(SNR_GratingDown) THEN
	Error_GratingDown:=TRUE;
END_IF;

//伺服回運轉中上光柵異常
IF (Ax_X.bHoming OR Ax_Y.bHoming OR Ax_X.pbSerchHome OR Ax_Y.pbSerchHome OR Ax_X.pbMoveAbs OR Ax_Y.pbMoveAbs  ) AND  NOT(SNR_GratingUP) THEN
	Ax_X.pbMoveAbs:=FALSE;
	Ax_Y.pbMoveAbs:=FALSE;
	Ax_X.pbSerchHome:=FALSE;
	Ax_Y.pbSerchHome:=FALSE;
	Error_GratingUP:=TRUE;
END_IF;
//伺服回運轉中下光柵異常
IF(Ax_X.bHoming OR Ax_Y.bHoming OR Ax_X.pbSerchHome OR Ax_Y.pbSerchHome OR Ax_X.pbMoveAbs OR Ax_Y.pbMoveAbs  ) AND  NOT(SNR_GratingDown) THEN
	Ax_X.pbMoveAbs:=FALSE;
	Ax_Y.pbMoveAbs:=FALSE;
	Ax_X.pbSerchHome:=FALSE;
	Ax_Y.pbSerchHome:=FALSE;
	Error_GratingDown:=TRUE;
END_IF;

(*磁簧開關異常*)
Error_LS_Status:=Error_LS_FixBack OR Error_LS_FixOut OR
                            Error_LS_UpDownBack OR Error_LS_UpDownOut;
							
//伺服異常
Error_Servo:=Error_Servo_X OR Error_Servo_Y OR Servo_OUT_Error;

//光柵異常
Error_Grating_Status:=Error_Check_GratingDown OR Error_Check_GratingUP OR
                                   Error_GratingDown OR   Error_GratingUP;                               
											
//鎖付異常
F_TRIG_2(Clk:=MachineRunStatus);
IF F_TRIG_2.Q AND NOT(Type_Data=10) AND (Screw_NG[4] OR Screw_NG[1]  OR Screw_NG[2]  OR Screw_NG[3] OR Screw_Float[1] OR Screw_Float[2] OR Screw_Float[3] OR Screw_Float[4] ) THEN
	Error_ScrewNG:=TRUE;
END_IF;				

//鎖付完成本體未置換
IF ScrewFinish AND PB_Start AND NOT(Type_Data=10) THEN
	Error_ChangeBodyNG:=TRUE;
END_IF;

IF NOT(SNR_CheckBody) OR(Type_Data=10) THEN
	ScrewFinish:=FALSE;
END_IF;

//X軸正極限異常
IF XP_OT AND State_Homed_MC  THEN
	Error_XP_OT:=TRUE;
	PB_ServoOn_X:=FALSE;
END_IF;
//X軸負極限異常
IF XN_OT  AND State_Homed_MC  THEN
	Error_XN_OT:=TRUE;
	PB_ServoOn_X:=FALSE;
END_IF;
//Y軸正極限異常
IF YP_OT  AND State_Homed_MC  THEN
	Error_YP_OT:=TRUE;
	PB_ServoOn_Y:=FALSE;
END_IF;
//Y軸負極限異常
IF YN_OT  AND State_Homed_MC  THEN
	Error_YN_OT:=TRUE;
	PB_ServoOn_Y:=FALSE;
END_IF;
IF NOT(XP_OT) AND NOT(XN_OT) AND NOT(YP_OT) AND NOT(YN_OT) AND (PB_HMI_RESRT OR PB_Reset ) THEN
	Error_XP_OT:=FALSE;
	Error_XN_OT:=FALSE;
	Error_YP_OT:=FALSE;
	Error_YN_OT:=FALSE;
	PB_ServoOn_X:=TRUE;
	PB_ServoOn_Y:=TRUE;
END_IF;

//外部取料完成
IF SystemReadyStatus AND (NOT( LS_ExternalStart) OR PB_ExternalStart) THEN
	ExternalStart_status:=TRUE;
END_IF;
IF LS_ExternalStart  AND ExternalStart_status THEN
	ReclaimerOK:=TRUE;
END_IF;
IF ReclaimerOK THEN
	ExternalStart_status:=FALSE;
END_IF;

//機器停機異常
ErrorStatus_MachineStop:=( Error_Servo AND NOT(Error_EStopPB)) OR  
											Error_Grating_Status OR					
											Error_SNR_AirSource OR
											Error_LS_Status ;
											
											//Error_ChangeBodyNG OR
											//Error_SNR_CheckBody;
											
(*復歸*)
IF PB_Reset  OR PB_HMI_RESRT  THEN
	Error_Check_GratingDown:=FALSE;
	Error_Check_GratingUP:=FALSE;
	Error_EStopPB:=FALSE;
    Error_GratingDown:=FALSE;
	Error_GratingUP:=FALSE;
	Error_SNR_AirSource:=FALSE;										
    Error_LS_FixBack:=FALSE;
	Error_LS_FixOut:=FALSE;
	Error_LS_UpDownBack:=FALSE;
	Error_LS_UpDownOut:=FALSE;
	Error_SNR_CheckBody:=FALSE;
	Error_Servo_X:=FALSE;
	Error_Servo_Y:=FALSE;
	Error_ChangeBodyNG:=FALSE;
	Error_ScrewNG:=FALSE;
	Error_ReclaimerOK:=FALSE;
END_IF;

//磁簧HMI對應
LS_UpDownBack1:=LS_UpDownBack;
LS_UpDownOut1:=LS_UpDownOut;
LS_FixBack1:=LS_FixBack;
LS_FixOut1:=LS_FixOut;
HMI_Servo_IN_Start:=Servo_IN_Start;

//原點復歸中
HMI_LT_ServoFinish:=LT_ServoFinish1 AND LT_ServoFinish2;
HMI_LT_ServoRuning:=LT_ServoRuning1 OR LT_ServoRuning2;
END_PROGRAM

PROGRAM Postion_Control
VAR
    AutoFlow : INT;
    InitFlow : INT;
    R_TRIG_1 : R_TRIG;
    R_TRIG_2 : R_TRIG;
    R_TRIG_3 : R_TRIG;
    R_TRIG_4 : R_TRIG;
    TON_1 : TON;
    F_TRIG_1 : F_TRIG;
    ii : INT;
    ErrorEstopStatus : BOOL;
END_VAR
VAR_EXTERNAL
    SystemReadyStatus : BOOL;
    AutoStatus : BOOL;
    PB_EStop : BOOL;
    Error_EStopPB : BOOL;
    PB_Start : BOOL;
    MachineRun : BOOL;
    ErrorStatus_MachineStop : BOOL;
    SNR_CheckBody : BOOL;
    SNR_GratingDown : BOOL;
    SNR_GratingUP : BOOL;
    PointData : INT;
    WorkPositionData : stWorkPositionData;
    Type_Data : INT;
    LS_UpDownBack : BOOL;
    Ax_X : stAxis;
    Ax_Y : stAxis;
    ScrewStartStatus : BOOL;
    LS_UpDownOut : BOOL;
    ScrewFinish : BOOL;
    LS_FixBack : BOOL;
    SOL_UpDownOut : BOOL;
    Error_Servo_X : BOOL;
    Error_Servo_Y : BOOL;
    Error_LS_Status : BOOL;
    PB_ServoX_Out : BOOL;
    PB_ServoX_Back : BOOL;
    PB_ServoY_Out : BOOL;
    PB_ServoY_Back : BOOL;
    SV_ServoXJogSpeed_R : REAL;
    SV_ServoYJogSpeed : LREAL;
    SV_ServoXJogSpeed : LREAL;
END_VAR
VAR_EXTERNAL CONSTANT
    MC_Axis000 : _sAXIS_REF;
    MC_Axis001 : _sAXIS_REF;
END_VAR
VAR_EXTERNAL
    PB_PostionGo : BOOL;
    Screw_OK : ARRAY[0..10] OF BOOL;
    Screw_NG : ARRAY[0..10] OF BOOL;
    PB_Reset : BOOL;
    State_Homed_MC : BOOL;
    MachineRunStatus : BOOL;
    Error_ScrewNG : BOOL;
    Error_ChangeBodyNG : BOOL;
    Error_SNR_CheckBody : BOOL;
    ReclaimerOK : BOOL;
    Error_ReclaimerOK : BOOL;
    PB_ExternalStart : BOOL;
    Screw_Float : ARRAY[0..10] OF BOOL;
END_VAR
(******************************************************************
程式:自動移位
作者:Andy_Wang
版本資訊:1.0.0		2017/9/16
PowerOn=0
Idle=1
清除資料點位歸零=2
檢查是否最終點=3
           |_______________________
           |									|
不是最終點 =4              是最終點=20
伺服位置寫入=5           伺服位置寫入=21
伺服啟動=6                   伺服啟動=22
伺服到位=7                   伺服到位=23
鎖付開始=8
鎖付中 =9
鎖付完成=10
point+1=11
******************************************************************)
//PowerOn=0
IF NOT(SystemReadyStatus) OR NOT(AutoStatus) OR Error_EStopPB THEN
	AutoFlow:=0;
END_IF;

//Idle=1
IF AutoFlow=0 AND AutoStatus AND NOT(Error_EStopPB) AND SystemReadyStatus THEN
	AutoFlow:=1;
END_IF;

IF AutoFlow=23 AND NOT(Ax_X.pbMoveAbs) AND NOT(Ax_Y.pbMoveAbs) AND NOT(MachineRun) THEN
	AutoFlow:=1;
END_IF;

//設備啟動
R_TRIG_1(Clk:=(AutoFlow=1  OR AutoFlow=4  OR AutoFlow=8) AND PB_Start  AND State_Homed_MC );
IF (AutoFlow=1 OR AutoFlow=4 OR AutoFlow=8 ) AND R_TRIG_1.Q  AND SNR_GratingDown  AND SNR_GratingUP AND NOT(ErrorStatus_MachineStop)  
	                                                  AND NOT(Ax_X.pbMoveAbs) AND NOT(Ax_Y.pbMoveAbs) AND NOT(ScrewFinish) 
													  and NOT(Error_ScrewNG) AND NOT(Error_ChangeBodyNG) AND NOT(Error_SNR_CheckBody)  THEN
MachineRun:=TRUE;
END_IF;

IF AutoFlow=0 OR Error_EStopPB OR ErrorStatus_MachineStop  OR PB_Reset OR AutoFlow=23 
	                    OR(Error_ScrewNG) OR(Error_ChangeBodyNG) OR (Error_SNR_CheckBody)  OR Error_ReclaimerOK  THEN
	MachineRun:=FALSE;
END_IF;
//外部取料異常
IF MachineRun AND NOT(ReclaimerOK) AND Type_Data<10 AND AutoFlow=1 AND NOT(PB_ExternalStart) THEN
	Error_ReclaimerOK:=TRUE;
END_IF;
//外部取料信號解除
IF    AutoFlow=23  OR (AutoFlow=1  AND NOT(SNR_CheckBody)) AND NOT(PB_ExternalStart)  THEN
	ReclaimerOK:=FALSE;
END_IF;

//設備運轉中
IF AutoFlow>1 THEN
	MachineRunStatus:=TRUE;
ELSE
	MachineRunStatus:=FALSE;
END_IF;


//清除資料點位設1=2 
R_TRIG_4(Clk:=MachineRun);
IF AutoFlow=1 AND R_TRIG_4.Q AND LS_UpDownBack AND  (ReclaimerOK OR Type_Data=10) AND   (SNR_CheckBody  OR Type_Data=10)  THEN
	AutoFlow:=2;
END_IF;
IF AutoFlow=2 THEN
	FOR ii:=1 TO 10 BY 1 DO
	    Screw_OK[ii]:=0;
		Screw_NG[ii]:=0;
		Screw_Float[ii]:=0;
	END_FOR;
	PointData:=1;
END_IF;

//檢查是否最終點=3
IF AutoFlow=2 AND PointData=1 AND Screw_OK[5]=Screw_OK[0] AND Screw_NG[5]=Screw_NG[0] AND Screw_Float[5]=Screw_Float[0]   THEN
	AutoFlow:=3;
END_IF;

//不是最終點 =4   
IF AutoFlow=3 AND NOT(WorkPositionData.FinialPoint[Type_Data,PointData]) AND PointData<10 THEN
	AutoFlow:=4;
END_IF;
 
// 伺服位置寫入=5  
IF AutoFlow=4 AND LS_UpDownBack AND MachineRun THEN
	AutoFlow:=5;
END_IF;
	
IF AutoFlow=5 THEN
	Ax_X.lrMoveAbsAddData:=WorkPositionData.ExPosition_X[Type_Data,PointData];
	Ax_Y.lrMoveAbsAddData:=WorkPositionData.ExPosition_Y[Type_Data,PointData];
	Ax_X.lrMoveAbsVelocity:=WorkPositionData.SV_AbsSpeed_X[Type_Data,PointData];
	Ax_Y.lrMoveAbsVelocity:=WorkPositionData.SV_AbsSpeed_Y[Type_Data,PointData];
END_IF;

//伺服啟動=6     
IF AutoFlow=5 AND (Ax_X.lrMoveAbsAddData=WorkPositionData.ExPosition_X[Type_Data,PointData])
	AND (Ax_Y.lrMoveAbsAddData=WorkPositionData.ExPosition_Y[Type_Data,PointData]) THEN
	AutoFlow:=6;
END_IF;

//伺服到位=7    
IF AutoFlow=6 AND TON_1.Q AND NOT(Ax_X.pbMoveAbs) AND NOT(Ax_Y.pbMoveAbs) THEN
	AutoFlow:=7;
END_IF;

//鎖付開始=8
IF AutoFlow=7 AND NOT(Ax_X.pbMoveAbs) AND NOT(Ax_Y.pbMoveAbs) THEN
	AutoFlow:=8;
END_IF;
IF AutoFlow=8 THEN
	ScrewStartStatus:=TRUE;
ELSE
		ScrewStartStatus:=FALSE;
END_IF;

//鎖付中 =9
IF AutoFlow=8 AND ScrewStartStatus AND LS_UpDownOut THEN
	AutoFlow:=9;
END_IF;

//鎖付完成=10
IF AutoFlow=9 AND LS_UpDownBack   THEN
	AutoFlow:=10;
END_IF;

//point+1=11
IF AutoFlow=10 AND LS_UpDownBack AND NOT(SOL_UpDownOut) THEN
	PointData:=PointData+1;
	AutoFlow:=11;
END_IF;
IF AutoFlow=11 THEN
	AutoFlow:=3;
END_IF;
//********************************************************************************************************

//是最終點=20
 IF AutoFlow=3 AND (WorkPositionData.FinialPoint[Type_Data,PointData]  OR PointData=10) THEN
	 AutoFlow:=20;
 END_IF;
 
  //伺服位置寫入=21
IF AutoFlow=20 AND LS_UpDownBack AND MachineRun THEN
	AutoFlow:=21;
END_IF;
	
IF AutoFlow=21 THEN
	Ax_X.lrMoveAbsAddData:=0;
	Ax_Y.lrMoveAbsAddData:=0;
	Ax_X.lrMoveAbsVelocity:=WorkPositionData.SV_AbsSpeed_X[Type_Data,PointData];
	Ax_Y.lrMoveAbsVelocity:=WorkPositionData.SV_AbsSpeed_Y[Type_Data,PointData];
END_IF;

//伺服啟動=22     
IF AutoFlow=21 AND (Ax_X.lrMoveAbsAddData=0)
	AND (Ax_Y.lrMoveAbsAddData=0) THEN
	AutoFlow:=22;
END_IF;

//伺服到位=23    
IF AutoFlow=22 AND TON_1.Q AND NOT(Ax_X.pbMoveAbs) AND NOT(Ax_Y.pbMoveAbs) THEN
	AutoFlow:=23;
	ScrewFinish:=TRUE;//鎖付完成信號
END_IF;
//清除鎖付完成信號
IF NOT(SNR_CheckBody) THEN
	ScrewFinish:=FALSE;
END_IF;
//***************************************************************************************************
TON_1(In:=AutoFlow=6 OR AutoFlow=22  , PT:=t#100ms);
R_TRIG_2(Clk:=AutoFlow=6 OR AutoFlow=22  );
IF R_TRIG_2.Q THEN
	Ax_X.pbMoveAbs:=TRUE;
	Ax_Y.pbMoveAbs:=TRUE;
END_IF;
//***************************************************************************************************
//異常
IF ErrorStatus_MachineStop  OR Error_EStopPB  THEN
	AutoFlow:=0;
	Ax_X.lrMoveAbsAddData:=0;
	Ax_Y.lrMoveAbsAddData:=0;
	Ax_X.pbMoveAbs:=FALSE;
	Ax_Y.pbMoveAbs:=FALSE;
END_IF;
//***************************************************************************************************
//X伺服手動出
Ax_X.pbJOGForward:=Ax_X.bServoOn AND PB_ServoX_Out AND NOT(AutoStatus) AND LS_UpDownBack AND NOT(SOL_UpDownOut)  ;
//X伺服手動歸
Ax_X.pbJOGBackward:=Ax_X.bServoOn AND PB_ServoX_Back AND NOT(AutoStatus) AND LS_UpDownBack AND NOT(SOL_UpDownOut)  ;
//Y伺服手動出
Ax_Y.pbJOGForward:=Ax_Y.bServoOn AND PB_ServoY_Out AND NOT(AutoStatus) AND LS_UpDownBack AND NOT(SOL_UpDownOut)  ;
//Y伺服手動歸
Ax_Y.pbJOGBackward:=Ax_Y.bServoOn AND PB_ServoY_Back AND NOT(AutoStatus) AND LS_UpDownBack AND NOT(SOL_UpDownOut)  ;
Ax_X.lrMoveJogVelocity:=SV_ServoXJogSpeed;
Ax_Y.lrMoveJogVelocity:=SV_ServoYJogSpeed;
//***************************************************************************************************
(*定位控制*)
R_TRIG_3(Clk:=PB_PostionGo AND NOT(AutoStatus) AND Ax_X.bServoOn AND Ax_Y.bServoOn AND MC_Axis000.Details.Homed AND MC_Axis001.Details.Homed);
IF R_TRIG_3.Q THEN
	Ax_X.lrMoveAbsAddData:=WorkPositionData.ExPosition_X[Type_Data,PointData];
	Ax_Y.lrMoveAbsAddData:=WorkPositionData.ExPosition_Y[Type_Data,PointData];
	Ax_X.lrMoveAbsVelocity:=WorkPositionData.SV_AbsSpeed_X[Type_Data,PointData];
	Ax_Y.lrMoveAbsVelocity:=WorkPositionData.SV_AbsSpeed_Y[Type_Data,PointData];
	IF  (Ax_X.lrMoveAbsAddData=WorkPositionData.ExPosition_X[Type_Data,PointData])
	AND (Ax_Y.lrMoveAbsAddData=WorkPositionData.ExPosition_Y[Type_Data,PointData]) THEN
	Ax_X.pbMoveAbs:=TRUE;
	Ax_Y.pbMoveAbs:=TRUE;
	END_IF;
END_IF;
//到達位置
IF Ax_X.bMoveAbsDone OR NOT(PB_EStop) OR ErrorStatus_MachineStop THEN
		Ax_X.pbMoveAbs:=FALSE;
END_IF;

IF Ax_Y.bMoveAbsDone OR NOT(PB_EStop)  OR ErrorStatus_MachineStop THEN
		Ax_Y.pbMoveAbs:=FALSE;
END_IF;	
END_PROGRAM

PROGRAM PR_fix
VAR
    AutoFlow : INT;
    interlockfixback : BOOL;
    interlockfixeout : BOOL;
    R_TRIG_1 : R_TRIG;
    R_TRIG_2 : R_TRIG;
    R_TRIG_3 : R_TRIG;
    R_TRIG_4 : R_TRIG;
    fixStatus : BOOL;
    InitFlow : INT;
    F_TRIG_1 : F_TRIG;
END_VAR
VAR_EXTERNAL
    SystemReadyStatus : BOOL;
    AutoStatus : BOOL;
    Error_EStopPB : BOOL;
    MachineRun : BOOL;
    LS_FixOut : BOOL;
    LS_UpDownBack : BOOL;
    LS_FixBack : BOOL;
    SOL_FixBack : BOOL;
    PB_EStop : BOOL;
    Error_LS_FixBack : BOOL;
    Error_LS_FixOut : BOOL;
    LS_UpDownOut : BOOL;
    SOL_UpDownOut : BOOL;
    PB_FixBack : BOOL;
    SOL_FixOut : BOOL;
    PB_FixOut : BOOL;
    ErrorStatus_MachineStop : BOOL;
    WorkPositionData : stWorkPositionData;
    Type_Data : INT;
    PointData : INT;
    ScrewFinish : BOOL;
    SNR_CheckBody : BOOL;
    ReclaimerOK : BOOL;
END_VAR
(******************************************************************
程式:旋轉壓制
作者:Andy_Wang
版本資訊:1.0.0		2017/9/16
PowerOn=0
Idle=1
壓制出=2
壓制歸=3
******************************************************************)
//PowerOn=0
IF NOT(SystemReadyStatus) OR NOT(AutoStatus) OR Error_EStopPB THEN
	AutoFlow:=0;
END_IF;

//Idle=1
IF AutoFlow=0 AND AutoStatus AND NOT(Error_EStopPB) AND SystemReadyStatus THEN
	AutoFlow:=1;
END_IF;
IF AutoFlow=3 AND LS_FixBack AND NOT(SOL_FixBack) THEN
	AutoFlow:=1;
END_IF;

R_TRIG_3(Clk:=MachineRun AND NOT(ScrewFinish) AND SNR_CheckBody  );
//壓制出=2
IF AutoFlow=1 AND R_TRIG_3.Q  AND NOT(Type_Data=10) AND ReclaimerOK  THEN
	AutoFlow:=2;
END_IF;
IF AutoFlow=2 AND LS_FixOut AND WorkPositionData.FinialPoint[Type_Data,PointData] THEN
	AutoFlow:=3;
END_IF;

//***************************************************************************************************
//異常
IF ErrorStatus_MachineStop OR Error_EStopPB  THEN
	AutoFlow:=0;
	SOL_FixBack:=FALSE;
	SOL_FixOut:=FALSE;
END_IF;
//***************************************************************************************************
(*手動*)
(*壓制電磁閥*)
interlockfixback:=LS_UpDownBack AND NOT(SOL_UpDownOut);
interlockfixeout:=LS_UpDownBack AND NOT(SOL_UpDownOut);
R_TRIG_1(CLK:=PB_FixBack AND NOT(AutoStatus));
IF (R_TRIG_1.Q  OR AutoFlow=3  OR InitFlow=3 ) AND interlockfixback THEN
	SOL_FixBack:=TRUE;
	SOL_FixOut:=FALSE;
END_IF;
IF LS_FixBack THEN
	SOL_FixBack:=FALSE;
END_IF;
R_TRIG_2(CLK:=PB_FixOut AND NOT(AutoStatus));
IF (R_TRIG_2.Q  OR AutoFlow=2) AND interlockfixeout THEN
	SOL_FixBack:=FALSE;
	SOL_FixOut:=TRUE;
END_IF;
IF LS_FixOut THEN
	SOL_FixOut:=FALSE;
END_IF;
END_PROGRAM

PROGRAM 鎖付程式
VAR
    AutoFlow : INT;
    InitFlow : INT;
    intScrewData : INT;
    R_TRIG_1 : R_TRIG;
    R_TRIG_2 : R_TRIG;
    R_TRIG_3 : R_TRIG;
    R_TRIG_4 : R_TRIG;
    F_TRIG_1 : F_TRIG;
    TON_1 : TON;
    TON_2 : TON;
    TON_3 : TON;
    TON_4 : TON;
    interlockUpDownback : BOOL;
    interlockUpDownOut : BOOL;
    ServoStartStatus : BOOL;
END_VAR
VAR_EXTERNAL
    SystemReadyStatus : BOOL;
    AutoStatus : BOOL;
    Error_EStopPB : BOOL;
    ScrewStartStatus : BOOL;
    Ax_X : stAxis;
    Ax_Y : stAxis;
    MachineRun : BOOL;
    WorkPositionData : stWorkPositionData;
    Type_Data : INT;
    PointData : INT;
    Servo_IN_Start : BOOL;
    Servo_OUT_NOK : BOOL;
    Servo_OUT_OK : BOOL;
    SNR_Float : BOOL;
    ScrewFinish : BOOL;
    Screw_OK : ARRAY[0..10] OF BOOL;
    Screw_NG : ARRAY[0..10] OF BOOL;
    PB_EStop : BOOL;
    Error_LS_FixBack : BOOL;
    Error_LS_FixOut : BOOL;
    Error_LS_Status : BOOL;
    LS_FixOut : BOOL;
    SOL_FixOut : BOOL;
    PB_FixBack : BOOL;
    PB_UpDownBack : BOOL;
    SOL_UpDownBack : BOOL;
    SOL_UpDownOut : BOOL;
    LS_FixBack : BOOL;
    LS_UpDownBack : BOOL;
    PB_UpDownOut : BOOL;
    LS_UpDownOut : BOOL;
    ErrorStatus_MachineStop : BOOL;
    Servo_IN_TorqueBit0 : BOOL;
    Servo_IN_TorqueBit1 : BOOL;
    Servo_IN_TorqueBit2 : BOOL;
    Servo_IN_TorqueBit3 : BOOL;
    PB_ScrewStart : BOOL;
    HMI_SV_Screw_Data : INT;
    OK_Count : DINT;
    AllOK_Count : DINT;
    PB_ResetOk_Count : BOOL;
    Screw_Float : ARRAY[0..10] OF BOOL;
END_VAR
(******************************************************************
程式:鎖螺絲
作者:Andy_Wang
版本資訊:1.0.0		2017/9/16
PowerOn=0
Idle=1
鎖付組別搬移=2
向下=3
起子運轉中=4
起子停止=5
浮鎖檢查=6
向上=7
******************************************************************)
//PowerOn=0
IF NOT(SystemReadyStatus) OR NOT(AutoStatus) OR Error_EStopPB THEN
	AutoFlow:=0;
END_IF;

//Idle=1
IF AutoFlow=0 AND AutoStatus AND NOT(Error_EStopPB) AND SystemReadyStatus THEN
	AutoFlow:=1;
END_IF;

IF AutoFlow=7 AND LS_UpDownBack   THEN
	AutoFlow:=1;
END_IF;

//鎖付組別搬移=2
IF AutoFlow=1 AND ScrewStartStatus AND NOT(Ax_X.pbMoveAbs) AND NOT(Ax_Y.pbMoveAbs) AND MachineRun AND (LS_FixOut OR Type_Data=10) THEN
	AutoFlow:=2;
END_IF;
IF AutoFlow=2 THEN
	intScrewData:=WorkPositionData.ScrewData[Type_Data,PointData];
	Screw_NG[PointData]:=FALSE;
	Screw_OK[PointData]:=FALSE;
	Screw_Float[PointData]:=FALSE;
END_IF;

//向下=3
IF AutoFlow=2 AND intScrewData=WorkPositionData.ScrewData[Type_Data,PointData] AND NOT(Screw_NG[PointData]) AND NOT(Screw_OK[PointData]) AND NOT(Screw_Float[PointData])  THEN
	AutoFlow:=3;
END_IF;

//起子運轉中=4
IF AutoFlow=3 AND NOT(Servo_OUT_NOK) AND NOT(Servo_OUT_OK) AND Servo_IN_Start THEN
	AutoFlow:=4;
END_IF;

//起子停止=5
IF AutoFlow=4 AND (Servo_OUT_NOK  OR Servo_OUT_OK )  THEN
	AutoFlow:=5;
END_IF;

IF AutoFlow=5 AND NOT(Servo_IN_Start)  AND  NOT(ScrewStartStatus) THEN 
	AutoFlow:=6;
END_IF;
//浮鎖檢查=6
TON_1(In:=AutoFlow=6  AND SNR_Float AND Servo_OUT_OK  , PT:=t#100ms);
TON_2(In:=AutoFlow=6  AND not(SNR_Float) AND Servo_OUT_OK  , PT:=t#500ms);
TON_4(In:=AutoFlow=6  AND  Servo_OUT_NOK  , PT:=t#100ms);
IF AutoFlow=6 AND TON_1.Q THEN
	Screw_OK[PointData]:=TRUE;       //鎖螺絲OK
END_IF;
IF AutoFlow=6 AND TON_4.Q    THEN
	Screw_NG[PointData]:=TRUE;      //鎖螺絲NG
END_IF;
IF AutoFlow=6 AND TON_2.Q    THEN
	Screw_Float[PointData]:=TRUE;      //浮鎖檢查NG
END_IF;

//向上=7
IF AutoFlow=6 AND (Screw_OK[PointData] OR Screw_NG[PointData] OR Screw_Float[PointData] ) THEN
	AutoFlow:=7;
END_IF;
R_TRIG_4(Clk:=AutoFlow=7 );
IF  AutoFlow=7 AND   Screw_OK[1] AND Screw_OK[2] AND Screw_OK[3] AND Screw_OK[4] AND R_TRIG_4.Q THEN
	OK_Count:=OK_Count+1;
	AllOK_Count:=AllOK_Count+1;
END_IF;
TON_3(In:=PB_ResetOk_Count  , PT:=t#2S);
IF TON_3.Q THEN
	OK_Count:=0;
END_IF;


//***************************************************************************************************
//異常
IF ErrorStatus_MachineStop  OR Error_EStopPB THEN
	AutoFlow:=0;
	Servo_IN_Start:=FALSE;
	SOL_UpDownBack:=FALSE;
	SOL_UpDownOut:=FALSE;
END_IF;
//***************************************************************************************************
(*手動*)
(*上下電磁閥歸*)
interlockUpDownback:=TRUE;
interlockUpDownOut:=NOT(Ax_X.pbMoveAbs) AND NOT(Ax_Y.pbMoveAbs);
R_TRIG_1(CLK:=PB_UpDownBack AND NOT(AutoStatus));
R_TRIG_2(CLK:=PB_UpDownOut AND NOT(AutoStatus));
IF (R_TRIG_1.Q  OR AutoFlow=7 OR InitFlow=2  ) AND interlockUpDownback THEN
	SOL_UpDownBack:=TRUE;
	SOL_UpDownOut:=FALSE;
END_IF;
IF LS_UpDownBack THEN
SOL_UpDownBack:=FALSE;
END_IF;
(*上下電磁閥出*)
IF (R_TRIG_2.Q  OR AutoFlow=3) AND interlockUpDownOut THEN
	SOL_UpDownBack:=FALSE;
	SOL_UpDownOut:=TRUE;
END_IF;
IF LS_UpDownOut THEN
SOL_UpDownOut:=FALSE;
END_IF;
//日東起子啟動
R_TRIG_3(CLK:=PB_ScrewStart AND NOT(AutoStatus));
IF ((R_TRIG_3.Q  AND NOT(ServoStartStatus)) OR AutoFlow=3 ) THEN
		Servo_IN_Start:=TRUE;
END_IF;
IF ((R_TRIG_3.Q  AND ServoStartStatus) OR AutoFlow=5 OR InitFlow=2 ) THEN
Servo_IN_Start:=FALSE;
END_IF;
ServoStartStatus:=Servo_IN_Start;

(*************************************************************************
程序名稱:RESET流程
作者:Andy_Wang
版本,日期,版本資訊:
1.0.0	2017/9/17		初始版本
PowerOn=0
Idle=1
上下回=2
*************************************************************************)
//PowerOn=0
IF NOT(SystemReadyStatus) THEN
	InitFlow:=0;
END_IF;
//Idle=1
IF InitFlow=0 AND SystemReadyStatus THEN
	InitFlow:=1;
END_IF;
IF InitFlow=2  AND LS_UpDownBack  AND NOT(SOL_UpDownBack)  AND NOT(Servo_IN_Start) THEN
	InitFlow:=1;
END_IF;
F_TRIG_1(Clk:=ErrorStatus_MachineStop );

//上下回=2
IF F_TRIG_1.Q AND InitFlow=1   THEN
	InitFlow:=2;
END_IF;
(*日東-Program*)
CASE HMI_SV_Screw_Data OF
	0:
	Servo_IN_TorqueBit0:=FALSE;
	Servo_IN_TorqueBit1:=FALSE;
	Servo_IN_TorqueBit2:=FALSE;
	Servo_IN_TorqueBit3:=FALSE;
	1:
	Servo_IN_TorqueBit0:=TRUE;
	Servo_IN_TorqueBit1:=FALSE;
	Servo_IN_TorqueBit2:=FALSE;
	Servo_IN_TorqueBit3:=FALSE;
	2:
	Servo_IN_TorqueBit0:=FALSE;
	Servo_IN_TorqueBit1:=TRUE;
	Servo_IN_TorqueBit2:=FALSE;
	Servo_IN_TorqueBit3:=FALSE;
	3:
	Servo_IN_TorqueBit0:=TRUE;
	Servo_IN_TorqueBit1:=TRUE;
	Servo_IN_TorqueBit2:=FALSE;
	Servo_IN_TorqueBit3:=FALSE;
	4:
	Servo_IN_TorqueBit0:=FALSE;
	Servo_IN_TorqueBit1:=FALSE;
	Servo_IN_TorqueBit2:=TRUE;
	Servo_IN_TorqueBit3:=FALSE;
	5:
	Servo_IN_TorqueBit0:=TRUE;
	Servo_IN_TorqueBit1:=FALSE;
	Servo_IN_TorqueBit2:=TRUE;
	Servo_IN_TorqueBit3:=FALSE;
	6:
	Servo_IN_TorqueBit0:=FALSE;
	Servo_IN_TorqueBit1:=TRUE;
	Servo_IN_TorqueBit2:=TRUE;
	Servo_IN_TorqueBit3:=FALSE;
	7:
	Servo_IN_TorqueBit0:=TRUE;
	Servo_IN_TorqueBit1:=TRUE;
	Servo_IN_TorqueBit2:=TRUE;
	Servo_IN_TorqueBit3:=FALSE;
	8:
	Servo_IN_TorqueBit0:=FALSE;
	Servo_IN_TorqueBit1:=FALSE;
	Servo_IN_TorqueBit2:=FALSE;
	Servo_IN_TorqueBit3:=TRUE;
	9:
	Servo_IN_TorqueBit0:=TRUE;
	Servo_IN_TorqueBit1:=FALSE;
	Servo_IN_TorqueBit2:=FALSE;
	Servo_IN_TorqueBit3:=TRUE;
	10:
	Servo_IN_TorqueBit0:=FALSE;
	Servo_IN_TorqueBit1:=TRUE;
	Servo_IN_TorqueBit2:=FALSE;
	Servo_IN_TorqueBit3:=TRUE;
	11:
	Servo_IN_TorqueBit0:=TRUE;
	Servo_IN_TorqueBit1:=TRUE;
	Servo_IN_TorqueBit2:=FALSE;
	Servo_IN_TorqueBit3:=TRUE;
	12:
	Servo_IN_TorqueBit0:=FALSE;
	Servo_IN_TorqueBit1:=FALSE;
	Servo_IN_TorqueBit2:=TRUE;
	Servo_IN_TorqueBit3:=TRUE;
	13:
	Servo_IN_TorqueBit0:=TRUE;
	Servo_IN_TorqueBit1:=FALSE;
	Servo_IN_TorqueBit2:=TRUE;
	Servo_IN_TorqueBit3:=TRUE;
	14:
	Servo_IN_TorqueBit0:=FALSE;
	Servo_IN_TorqueBit1:=TRUE;
	Servo_IN_TorqueBit2:=TRUE;
	Servo_IN_TorqueBit3:=TRUE;
	15:
	Servo_IN_TorqueBit0:=TRUE;
	Servo_IN_TorqueBit1:=TRUE;
	Servo_IN_TorqueBit2:=TRUE;
	Servo_IN_TorqueBit3:=TRUE;
END_CASE;
END_PROGRAM

PROGRAM 異常回0點
VAR
    InitFlow : INT;
    R_TRIG_1 : R_TRIG;
    R_TRIG_2 : R_TRIG;
    TON_1 : TON;
    TON_2 : TON;
    F_TRIG_1 : F_TRIG;
END_VAR
VAR_EXTERNAL
    SystemReadyStatus : BOOL;
    PB_Set_Homed : BOOL;
    SOL_UpDownBack : BOOL;
    SOL_UpDownOut : BOOL;
    Servo_IN_Start : BOOL;
    LS_UpDownBack : BOOL;
    SOL_FixBack : BOOL;
    SOL_FixOut : BOOL;
    LS_FixBack : BOOL;
    Ax_X : stAxis;
    Ax_Y : stAxis;
    WorkPositionData : stWorkPositionData;
    Type_Data : INT;
    PointData : INT;
    Manual2AutoFlag : BOOL;
    Error_EStopPB : BOOL;
    AutoStatus : BOOL;
    State_Homed_MC : BOOL;
    ErrorStatus_MachineNonStop : BOOL;
    ErrorStatus_MachineStop : BOOL;
    PB_EStop : BOOL;
    State_Homing_MC : BOOL;
    State_Homed_Y : BOOL;
    LT_ServoFinish1 : BOOL;
    LT_ServoRuning1 : BOOL;
    Error_ScrewNG : BOOL;
    PB_ServoOn_X : BOOL;
    PB_ServoOn_Y : BOOL;
END_VAR
(*************************************************************************
程序名稱:伺服回0點流程
作者:Andy_Wang
版本,日期,版本資訊:
1.0.0	2017/9/17		初始版本
PowerOn=0
Idle=1
上下回=2
type<10壓制回=3---------------------type=10壓制不作動=7
伺服移至0點=4
伺服起動=5
伺服到位=6
*************************************************************************)
//PowerOn=0
IF NOT(SystemReadyStatus) THEN
	InitFlow:=0;
END_IF;
//Idle=1
IF InitFlow=0 AND SystemReadyStatus THEN
	InitFlow:=1;
END_IF;
IF InitFlow=6 THEN
	InitFlow:=1;
END_IF;
//伺服回歸完成信號
IF InitFlow<=1 THEN
	LT_ServoFinish1:=TRUE;
ELSE
	LT_ServoFinish1:=FALSE;
END_IF;
//伺服回歸中信號
IF InitFlow>1 THEN
	LT_ServoRuning1:=TRUE;
ELSE
	LT_ServoRuning1:=FALSE;
END_IF;


//上下回=2
F_TRIG_1(Clk:=ErrorStatus_MachineStop AND State_Homed_MC   );
R_TRIG_1(Clk:=PB_Set_Homed OR Manual2AutoFlag AND (Ax_X.lrCurrentPosition<>0 OR Ax_Y.lrCurrentPosition<>0));
IF (R_TRIG_1.Q  OR F_TRIG_1.Q) AND InitFlow=1  THEN
	SOL_UpDownBack:=TRUE;
	SOL_UpDownOut:=FALSE;
	Servo_IN_Start:=FALSE;
	PB_ServoOn_X:=TRUE;
	PB_ServoOn_Y:=TRUE;
	InitFlow:=2;
END_IF;

//type<10壓制回=3
IF InitFlow=2 AND LS_UpDownBack AND NOT(Servo_IN_Start) AND NOT(SOL_UpDownBack) AND Type_Data<10  THEN
	SOL_FixBack:=TRUE;
	SOL_FixOut:=FALSE;
	InitFlow:=3;
END_IF;
//type=10壓制不作動=7
IF InitFlow=2 AND LS_UpDownBack AND NOT(Servo_IN_Start) AND NOT(SOL_UpDownBack) AND Type_Data=10  THEN
	InitFlow:=7;
END_IF;
//伺服移至0點=4
IF (InitFlow=3 AND LS_FixBack AND NOT(SOL_FixBack))  OR (InitFlow=7) THEN
	Ax_X.lrMoveAbsAddData:=0;
	Ax_Y.lrMoveAbsAddData:=0;
	Ax_X.lrMoveAbsVelocity:=70;
	Ax_Y.lrMoveAbsVelocity:=70;
	InitFlow:=4;
END_IF;
TON_2(In:=InitFlow=4, PT:=t#300ms);
//伺服起動=5
IF InitFlow=4 AND Ax_X.lrMoveAbsAddData=0  AND Ax_Y.lrMoveAbsAddData=0 AND TON_2.Q  THEN
	InitFlow:=5;
END_IF;

//伺服到位=6
TON_1(In:=InitFlow=5, PT:=t#100ms);
IF InitFlow=5 AND NOT(Ax_X.pbMoveAbs) AND NOT(Ax_Y.pbMoveAbs)  AND TON_1.Q THEN
InitFlow:=6;
END_IF;

R_TRIG_2(Clk:=InitFlow=5);
IF R_TRIG_2.Q THEN
Ax_X.pbMoveAbs:=TRUE;
Ax_Y.pbMoveAbs:=TRUE;
END_IF;
//到達位置
IF Ax_X.bMoveAbsDone OR NOT(PB_EStop) OR ErrorStatus_MachineStop THEN
		Ax_X.pbMoveAbs:=FALSE;
END_IF;

IF Ax_Y.bMoveAbsDone OR NOT(PB_EStop)  OR ErrorStatus_MachineStop THEN
		Ax_Y.pbMoveAbs:=FALSE;
END_IF;	

//異常
IF ErrorStatus_MachineStop  OR Error_EStopPB  THEN
	InitFlow:=0;
	Ax_X.pbMoveAbs:=FALSE;
    Ax_Y.pbMoveAbs:=FALSE;
	Ax_X.lrMoveAbsAddData:=0;
	Ax_Y.lrMoveAbsAddData:=0;
END_IF;
	
END_PROGRAM

PROGRAM 系統初始
VAR
    SystemInitFlow : INT := 0;
    TON_1 : TON;
    TON_2 : TON;
    TON_3 : TON;
    TON_4 : TON;
    R_TRIG_3 : R_TRIG;
    BzTimer : bool;
    InitFlow : int;
    F_TRIG_1 : F_TRIG;
END_VAR
VAR_EXTERNAL
    AutoStatus : BOOL;
    SystemReadyStatus : BOOL;
    PB_EStop : BOOL;
    Error_EStopPB : BOOL;
END_VAR
VAR_EXTERNAL CONSTANT
    MC_Axis000 : _sAXIS_REF;
    MC_Axis001 : _sAXIS_REF;
END_VAR
VAR_EXTERNAL
    PB_ServoOn_X : BOOL;
    PB_ServoOn_Y : BOOL;
    Ax_X : stAxis;
    Ax_Y : stAxis;
    SOL_UpDownBack : BOOL;
    LS_UpDownBack : BOOL;
    SOL_FixBack : BOOL;
    LS_FixBack : BOOL;
    Manual2AutoFlag : BOOL;
    BZ : BOOL;
    ErrorStatus_MachineStop : BOOL;
    MachineRun : BOOL;
    RL : BOOL;
    GL : BOOL;
    YL : BOOL;
    Error_GratingUP : BOOL;
    Error_GratingDown : BOOL;
    Error_Grating_Status : BOOL;
    Error_Servo : BOOL;
    Error_SNR_AirSource : BOOL;
    Error_LS_Status : BOOL;
    PB_Reset : BOOL;
    MachineRunStatus : BOOL;
    ErrorStatus_MachineNonStop : BOOL;
    State_Homed_MC : BOOL;
    Error_SNR_CheckBody : BOOL;
    Error_ScrewNG : BOOL;
    Error_ChangeBodyNG : BOOL;
    PB_HMI_BzStpo : BOOL;
    Error_XN_OT : BOOL;
    Error_XP_OT : BOOL;
    Error_YN_OT : BOOL;
    Error_YP_OT : BOOL;
    Error_ReclaimerOK : BOOL;
    Type_Data : INT;
END_VAR
(******************************************************************
程式:系統初始化
作者:Andy_Wang
版本資訊:1.0.0		2017/9/16

全部狀態RESET=0
伺服上電=1
伺服未回HOME=2
伺服Servo on=3
伺服Ready=4
上下回=5
壓制回=6
伺服X軸Serch Home=7
伺服X軸Serch Home中=8
伺服X軸Serch Home完成=9
伺服Y軸Serch Home=10
伺服Y軸Serch Home中=11
伺服Y軸Serch Home完成=12
自動SET=13
系統READY SET=14
Init完成=15
******************************************************************)
//全部狀態RESET=0
IF P_First_Run  THEN
		SystemInitFlow:=0;
		AutoStatus:=FALSE;
		SystemReadyStatus:=FALSE;
END_IF;
//伺服上電=1
IF 	SystemInitFlow=0 AND PB_EStop AND NOT(Error_EStopPB) AND NOT(AutoStatus) 
AND NOT(SystemReadyStatus) AND MC_Axis000.DrvStatus.MainPower AND MC_Axis001.DrvStatus.MainPower THEN
SystemInitFlow:=1;
END_IF;

//伺服未回HOME=2
IF SystemInitFlow=1 AND NOT(MC_Axis000.Details.Homed) AND NOT(MC_Axis001.Details.Homed) THEN
	SystemInitFlow:=2;
END_IF;

//伺服回HOME=2
IF SystemInitFlow=1 AND MC_Axis000.Details.Homed AND MC_Axis001.Details.Homed THEN
	SystemInitFlow:=2;
END_IF;

//伺服Servo on=3
IF SystemInitFlow=2 THEN
	SystemInitFlow:=3;
END_IF;

IF SystemInitFlow=3 THEN
	PB_ServoOn_X:=TRUE;
	PB_ServoOn_Y:=TRUE;
END_IF;

//伺服Ready=4
IF SystemInitFlow=3 AND Ax_X.bServoOn AND Ax_Y.bServoOn AND MC_Axis000.DrvStatus.Ready AND MC_Axis001.DrvStatus.Ready THEN
	SystemInitFlow:=4;
END_IF;

//上下回=5
IF SystemInitFlow=4 THEN
	SystemInitFlow:=5;
END_IF;
IF SystemInitFlow=5 THEN
	SOL_UpDownBack:=TRUE;
END_IF;
IF LS_UpDownBack THEN
	SOL_UpDownBack:=FALSE;
END_IF;

//壓制回=6
IF SystemInitFlow=5 AND LS_UpDownBack AND NOT(SOL_UpDownBack) THEN
	SystemInitFlow:=6;
END_IF;
IF SystemInitFlow=6 AND Type_Data<10 THEN
	SOL_FixBack:=TRUE;
END_IF;
IF LS_FixBack THEN
	SOL_FixBack:=FALSE;
END_IF;

//伺服X軸Serch Home=7
TON_3(In:=SystemInitFlow=6 AND Ax_X.bServoOn AND Ax_Y.bServoOn  , PT:=T#1000ms);
IF  SystemInitFlow=6 AND LS_UpDownBack AND (LS_FixBack OR Type_Data=10) AND NOT(SOL_FixBack) AND TON_3.Q THEN
	SystemInitFlow:=7;
END_IF;
IF SystemInitFlow=7 THEN
	Ax_X.pbSerchHome:=TRUE;
	Ax_Y.pbSerchHome:=TRUE;
END_IF;

//伺服X軸Serch Home中=8	
IF SystemInitFlow=7 AND Ax_X.bHoming THEN
	Ax_X.pbSerchHome:=FALSE;
END_IF;
//伺服X軸Serch Home中=8	
IF SystemInitFlow=7 AND Ax_Y.bHoming THEN
	Ax_Y.pbSerchHome:=FALSE;
END_IF;

IF SystemInitFlow=7 AND NOT(Ax_X.pbSerchHome) AND NOT(Ax_Y.pbSerchHome)  THEN
	SystemInitFlow:=8;
END_IF;
//伺服X軸Serch Home完成=9
IF SystemInitFlow=8 AND NOT(Ax_X.bHoming)  AND  NOT(Ax_Y.bHoming) THEN
	SystemInitFlow:=9;
END_IF;
//TON_4(In:=SystemInitFlow=9 AND Ax_Y.bServoOn , PT:=T#1000ms);
//伺服Y軸Serch Home=10
//IF SystemInitFlow=9 AND MC_Axis000.Details.Homed AND TON_4.Q THEN
//	SystemInitFlow:=10;
//END_IF;
//IF SystemInitFlow=10 THEN
//Ax_Y.pbSerchHome:=TRUE;
//END_IF;

//伺服Y軸Serch Home中=11
//IF SystemInitFlow=10 AND Ax_Y.bHoming THEN
	//Ax_Y.pbSerchHome:=FALSE;
//	SystemInitFlow:=11;
//END_IF;

//伺服Y軸Serch Home完成=12
//IF SystemInitFlow=11 AND NOT(Ax_Y.bHoming) THEN
//	SystemInitFlow:=12;
//END_IF;

//自動SET=13
IF SystemInitFlow=9 AND MC_Axis001.Details.Homed AND MC_Axis000.Details.Homed  THEN
	SystemInitFlow:=13;
END_IF;
IF SystemInitFlow=13 THEN
	AutoStatus:=TRUE;
END_IF;//系統READY SET=14
IF SystemInitFlow=13 AND AutoStatus THEN
	SystemInitFlow:=14;
END_IF;
IF SystemInitFlow=14 THEN
	SystemReadyStatus:=TRUE;
END_IF;

//Init完成=15
IF SystemInitFlow=14 AND SystemReadyStatus   THEN
	SystemInitFlow:=15;
END_IF;
//系統初始錯誤歸零
F_TRIG_1(Clk:=(Error_EStopPB OR ErrorStatus_MachineStop) AND NOT(State_Homed_MC));
IF SystemInitFlow<15 AND NOT(SystemReadyStatus)  AND F_TRIG_1.Q THEN
	SystemInitFlow:=4;
	Ax_X.pbSerchHome:=FALSE;
	Ax_Y.pbSerchHome:=FALSE;
END_IF;


//******************************************************************
//手動轉自動
R_TRIG_3(Clk:=AutoStatus, Q=>Manual2AutoFlag);
(******************************************************************
程式:燈號及蜂鳴器
作者:Andy Wang
版本資訊:1.0.0		2017/9/16
******************************************************************)
//設備運轉中(GL)
IF (MachineRun AND NOT(RL)) OR (MachineRunStatus AND BzTimer AND NOT(RL) )   (*OR (NOT(State_Homed_MC)  AND NOT(Error_EStopPB))*)  THEN
	GL:=TRUE;
ELSE
	GL:=FALSE;
END_IF;
//待機(YL)
IF AutoStatus AND  NOT(RL) AND NOT(GL) AND NOT(MachineRunStatus) AND NOT(ErrorStatus_MachineStop) AND NOT(Error_EStopPB)  THEN
	YL:=TRUE;
ELSE
	YL:=FALSE;
END_IF;
//異常(RL)
IF (Error_Grating_Status AND BzTimer)  OR  (Error_Servo  OR Error_SNR_AirSource OR Error_LS_Status OR Error_SNR_CheckBody  OR Error_ScrewNG  OR Error_ChangeBodyNG
                                                                                                  OR  Error_XN_OT OR Error_XP_OT OR Error_YN_OT  OR Error_YP_OT OR Error_ReclaimerOK ) THEN
	RL:=TRUE;
ELSE
	RL:=FALSE;
END_IF;
//蜂鳴器(BZ)
IF Error_EStopPB  AND NOT(PB_HMI_BzStpo) OR (BzTimer AND  NOT(PB_HMI_BzStpo) AND  (Error_Grating_Status  OR Error_Servo OR Error_SNR_AirSource  OR Error_LS_Status  OR Error_SNR_CheckBody  OR Error_ScrewNG  OR Error_ChangeBodyNG
                                                                                                                    OR  Error_XN_OT OR Error_XP_OT OR Error_YN_OT  OR Error_YP_OT OR Error_ReclaimerOK ) )  THEN
	BZ:=TRUE;
ELSE
	BZ:=FALSE;
END_IF;

TON_1(In:=not(BzTimer), PT:=T#1000ms);
IF TON_1.Q THEN
	BzTimer:=TRUE;
END_IF;
TON_2(In:=BzTimer, PT:=T#1000ms);
IF TON_2.Q THEN
	BzTimer:=FALSE;
END_IF;
END_PROGRAM

PROGRAM cycletime2
VAR
    test1 : BOOL;
    R_TRIG_1 : R_TRIG;
    R_TRIG_2 : R_TRIG;
    F_TRIG_1 : F_TRIG;
    TON_1 : TON;
    TON_2 : TON;
    TON_3 : TON;
    AutoFlow : INT;
    CycleTime0 : LINT;
    CycleTime1 : DINT;
END_VAR
VAR_EXTERNAL
    HMISV_CycleTime1 : DINT;
    HMISV_CycleTime2 : DINT;
    SystemReadyStatus : BOOL;
    MachineRun : BOOL;
    MachineRunStatus : BOOL;
END_VAR
(******************************************************************
程式:CycleTimer
作者:Andy_Wang
版本資訊:1.0.0		2017/9/16
PowerOn=0
Idle=1
儲存至前次加工時間=2
儲存完畢=3
計算值登錄至現在值=4
計時結束=5
       
******************************************************************)
IF NOT(SystemReadyStatus) THEN
	AutoFlow:=0;
END_IF;

IF AutoFlow=0  AND SystemReadyStatus THEN
	AutoFlow:=1;
END_IF;

IF AutoFlow=5  THEN
	AutoFlow:=1;
END_IF;

//儲存至前次加工時間=2
R_TRIG_1(Clk:=MachineRunStatus);
F_TRIG_1(Clk:=MachineRunStatus);
IF AutoFlow=1 AND R_TRIG_1.Q THEN
	HMISV_CycleTime2:=HMISV_CycleTime1;
	AutoFlow:=2;
END_IF;

//儲存完畢=3
TON_1(In:=AutoFlow=2, PT:=t#1ms);
IF AutoFlow=2 AND TON_1.Q AND HMISV_CycleTime2=HMISV_CycleTime1 THEN
	AutoFlow:=3;
END_IF;

//計算值登錄至現在值=4
IF AutoFlow=3 THEN
	AutoFlow:=4;
END_IF;

IF AutoFlow=4 THEN
	CycleTime1:=LINT_TO_DINT(CycleTime0);
	HMISV_CycleTime1:=CycleTime1;
	AutoFlow:=4;
END_IF;
	
//計時結束=5
IF  AutoFlow=4  AND F_TRIG_1.Q THEN
	AutoFlow:=5;
END_IF;

//數值換算
TON_2(In:=AutoFlow>2 AND AutoFlow<5   , PT:=t#500s);
CycleTime0:=TimeToSec(TON_2.ET);


	
END_PROGRAM

PROGRAM 原點復歸
VAR
    AutoFlow : INT;
    F_TRIG_1 : F_TRIG;
    Reset_Start : BOOL;
    EC_Error : BOOL;
    EC_Err_Level : UINT;
    EC_Err_Code : DWORD;
    MC_Error : BOOL;
    MC_Err_Level : UINT;
    MC_Err_Code : DWORD;
    EC_Stage : INT;
    ResetECError_instance : ResetECError;
    MC_Stage : INT;
    ResetMCError_instance : ResetMCError;
    TON_2 : TON;
    SystemInitFlow : INT := 0;
    TON_3 : TON;
END_VAR
VAR_EXTERNAL
    SystemReadyStatus : BOOL;
    Error_EStopPB : BOOL;
    State_Homed_MC : BOOL;
    Ax_X : stAxis;
    Ax_Y : stAxis;
END_VAR
VAR_EXTERNAL CONSTANT
    MC_Axis000 : _sAXIS_REF;
    MC_Axis001 : _sAXIS_REF;
END_VAR
VAR_EXTERNAL
    PB_ServoOn_X : BOOL;
    PB_ServoOn_Y : BOOL;
    SOL_UpDownBack : BOOL;
    LS_UpDownBack : BOOL;
    SOL_FixBack : BOOL;
    LS_FixBack : BOOL;
    AutoStatus : BOOL;
    ErrorStatus_MachineStop : BOOL;
    State_Homing_MC : BOOL;
    LT_ServoFinish2 : BOOL;
    LT_ServoRuning2 : BOOL;
    Type_Data : INT;
END_VAR
(******************************************************************
程式:原點復歸
作者:Andy_Wang
版本資訊:1.0.0		2017/9/16

Power_ON=0
IDLE=1
全部狀態RESET=2
PLC異常初始化開始=3
PLC初始化完成=4
伺服未回HOME=5
伺服Servo on=6
伺服Ready=7
上下回=8
壓制回=9
伺服XY軸Serch Home開始=10
伺服XY軸Serch Home中=11
伺服XY軸Serch Home完成=12
伺服XY軸完成=13

******************************************************************)
//Power_ON=0
IF NOT(SystemReadyStatus) THEN
	AutoFlow:=0;
END_IF;

//IDLE=1
IF AutoFlow=0 AND SystemReadyStatus THEN
	AutoFlow:=1;
END_IF;

IF AutoFlow=13  THEN
	AutoFlow:=1;
END_IF;

//伺服回歸完成信號
IF AutoFlow<=1 THEN
	LT_ServoFinish2:=TRUE;
ELSE
	LT_ServoFinish2:=FALSE;
END_IF;
//伺服回歸中信號
IF AutoFlow>1 THEN
	LT_ServoRuning2:=TRUE;
ELSE
	LT_ServoRuning2:=FALSE;
END_IF;

//全部狀態RESET=2
F_TRIG_1(Clk:=(Error_EStopPB OR ErrorStatus_MachineStop) AND NOT(State_Homed_MC));
IF AutoFlow=1 AND F_TRIG_1.Q   THEN
	AutoFlow:=2;
END_IF;
IF AutoFlow=2 THEN
	Ax_X.pbSerchHome:=FALSE;
	Ax_Y.pbSerchHome:=FALSE;
	Ax_X.pbMoveAbs:=FALSE;
	Ax_Y.pbMoveAbs:=FALSE;
	AutoStatus:=FALSE;
END_IF;

//PLC異常初始化開始=3
IF AutoFlow=2 AND NOT(Ax_X.pbSerchHome)  AND NOT(Ax_Y.pbSerchHome)  
	                     AND NOT(Ax_X.pbMoveAbs) AND NOT(Ax_Y.pbMoveAbs) AND NOT(AutoStatus) THEN
	AutoFlow:=3;
END_IF;
IF AutoFlow=3 THEN
	Reset_Start:=TRUE;
END_IF;

IF  AutoFlow=3  AND Reset_Start   THEN
	EC_Error:=GetECError(EC_Err_Level, EC_Err_Code); // EtherCAT 功能模块的控制器异常检测
    MC_Error:=GetMCError(MC_Err_Level, MC_Err_Code); // 运动控制功能模块的控制器异常检测
   IF (EC_Error=TRUE) THEN // 有EtherCAT 功能模块的控制器异常
  CASE EC_Stage OF
  0 : // 初始化
  ResetECError_instance(Execute:=FALSE);
  EC_Stage:=INT#1;
  1 : // EtherCAT 功能模块的控制器异常解除中
  ResetECError_instance(Execute:=TRUE);
  IF (ResetECError_instance.Done=TRUE) THEN
  EC_Stage:=INT#99; // 正常结束
  END_IF;
  IF (ResetECError_instance.Error=TRUE) THEN
  EC_Stage:=INT#98; // 异常结束
  END_IF;
  99 : // 正常结束时处理
  EC_Stage:=INT#0; 
  98 : // 异常结束时处理
  EC_Stage:=INT#0;
  END_CASE;
  END_IF;
  IF (MC_Error=TRUE) THEN // 有运动控制功能模块的控制器异常
  CASE MC_Stage OF
  0 : // 初始化
  ResetMCError_instance(Execute:=FALSE);
  MC_Stage:=INT#1;
  1 : // 运动控制功能模块的控制器异常解除中
  IF (EC_Error=FALSE) THEN
  ResetMCError_instance(Execute:=TRUE); // 全部从站复位
  IF (ResetMCError_instance.Done=TRUE) THEN
  MC_Stage:=INT#99; // 正常结束
  END_IF;
  IF ( (ResetMCError_instance.Error=TRUE) OR (ResetMCError_instance.Failure=TRUE) ) THEN
  MC_Stage:=INT#98; // 异常结束
  END_IF;
 END_IF;
  99 : // 正常结束时处理 
  MC_Stage:=INT#0;
  98 : // 异常结束时处理
  MC_Stage:=INT#0;
  END_CASE;
  END_IF;
  END_IF;
 // PLC初始化完成=4
TON_2(In:=AutoFlow=3 AND  NOT(EC_Error) AND NOT(MC_Error)  , PT:=T#3S );
IF AutoFlow=3 AND NOT(EC_Error) AND NOT(MC_Error) AND TON_2.Q THEN
	AutoFlow:=4;
	Reset_Start:=FALSE;
END_IF;

//伺服未回HOME=5
IF AutoFlow=4 AND NOT(Reset_Start) AND  ((NOT(MC_Axis000.Details.Homed) AND NOT(MC_Axis001.Details.Homed)) OR
	                              (MC_Axis000.Details.Homed AND MC_Axis001.Details.Homed) OR
								  (MC_Axis000.Details.Homed AND NOT(MC_Axis001.Details.Homed)) OR
								  (NOT(MC_Axis000.Details.Homed) AND MC_Axis001.Details.Homed))  THEN
	AutoFlow:=5;
END_IF;

//伺服Servo on=6
IF AutoFlow=5 THEN
	AutoFlow:=6;
END_IF;
IF AutoFlow=6 THEN
	PB_ServoOn_X:=TRUE;
	PB_ServoOn_Y:=TRUE;
END_IF;

//伺服Ready=7
IF AutoFlow=6 AND Ax_X.bServoOn AND Ax_Y.bServoOn AND MC_Axis000.DrvStatus.Ready AND MC_Axis001.DrvStatus.Ready THEN
	AutoFlow:=7;
END_IF;

//上下回=8
IF AutoFlow=7 THEN
	AutoFlow:=8;
END_IF;
IF AutoFlow=8 THEN
	SOL_UpDownBack:=TRUE;
END_IF;
IF LS_UpDownBack THEN
	SOL_UpDownBack:=FALSE;
END_IF;

//壓制回=9
IF AutoFlow=8 AND LS_UpDownBack AND NOT(SOL_UpDownBack) THEN
	AutoFlow:=9;
END_IF;
IF AutoFlow=9 AND NOT(Type_Data=10)THEN
	SOL_FixBack:=TRUE;
END_IF;
IF (LS_FixBack OR Type_Data=10)  THEN
	SOL_FixBack:=FALSE;
END_IF;

//伺服XY軸Serch Home開始=10
TON_3(In:=AutoFlow=9 AND Ax_X.bServoOn AND Ax_Y.bServoOn  , PT:=T#1000ms);
IF  AutoFlow=9 AND LS_UpDownBack AND (LS_FixBack OR Type_Data=10) AND NOT(SOL_FixBack) AND TON_3.Q THEN
	AutoFlow:=10;
END_IF;
IF AutoFlow=10 THEN
	Ax_X.pbSerchHome:=TRUE;
	Ax_Y.pbSerchHome:=TRUE;
END_IF;
//伺服XY軸Serch Home中=11
IF  AutoFlow=10 AND ((Ax_X.pbSerchHome OR Ax_X.bHoming OR MC_Axis000.Details.Homed )AND
                                     (Ax_Y.pbSerchHome  OR Ax_Y.bHoming OR MC_Axis001.Details.Homed))                             
									 THEN
	AutoFlow:=11;
END_IF;
IF AutoFlow=11 AND (Ax_X.bHoming  OR MC_Axis000.Details.Homed)  THEN
	Ax_X.pbSerchHome:=FALSE;
END_IF;
IF AutoFlow=11 AND (Ax_Y.bHoming OR MC_Axis001.Details.Homed)  THEN
	Ax_Y.pbSerchHome:=FALSE;
END_IF;

//伺服XY軸Serch Home完成=12
IF AutoFlow=11 AND MC_Axis001.Details.Homed AND MC_Axis000.Details.Homed 
	                       AND NOT(Ax_X.pbSerchHome) AND NOT(Ax_Y.pbSerchHome)   THEN
	AutoFlow:=12;
END_IF;
IF AutoFlow=12 THEN
	AutoStatus:=TRUE;
END_IF;

//伺服XY軸完成=13
IF AutoFlow=12 AND AutoStatus THEN
	AutoFlow:=13;
END_IF;
//******************************************************************
//異常
IF ErrorStatus_MachineStop  OR Error_EStopPB  THEN
	AutoFlow:=0;
	Ax_X.pbSerchHome:=FALSE;
	Ax_Y.pbSerchHome:=FALSE;
END_IF;
END_PROGRAM